# B&R Automation Studio project TD52 (part 144)

#### rtwtypes.h
```c
/********************************************************************
 * COPYRIGHT -- Bernecker + Rainer Industrie-Elektronik Ges.m.b.H.
 ********************************************************************
 * Program: J920_fric
 * File: rtwtypes.h
 * Author: 212348321
 * Created: Mon Jun 13 15:26:38 2016
 ********************************************************************
 * Header for program J920_fric
 ********************************************************************
 * Generated with B&R Automation Studio Target for Simulink V4.2
 * (ERT based)
 ********************************************************************/

#ifndef __RTWTYPES_H__
#define __RTWTYPES_H__
#ifndef TRUE
# define TRUE                          (1U)
#endif

#ifndef FALSE
# define FALSE                         (0U)
#endif

#ifndef __TMWTYPES__
#define __TMWTYPES__
#include <limits.h>

/*=======================================================================*
 * Target hardware information
 *   Device type: Intel->x86/Pentium
 *   Number of bits:     char:   8    short:   16    long:  32
 *                       long:  32
 *                       native word size:  32
 *   Byte ordering: LittleEndian
 *   Signed integer division rounds to: Zero
 *   Shift right on a signed integer as arithmetic shift: on
 *=======================================================================*/

/*=======================================================================*
 * Fixed width word size data types:                                     *
 *   int8_T, int16_T, int32_T     - signed 8, 16, or 32 bit integers     *
 *   uint8_T, uint16_T, uint32_T  - unsigned 8, 16, or 32 bit integers   *
 *   real32_T, real64_T           - 32 and 64 bit floating point numbers *
 *=======================================================================*/
typedef signed char int8_T;
typedef unsigned char uint8_T;
typedef short int16_T;
typedef unsigned short uint16_T;
typedef long int32_T;
typedef unsigned long uint32_T;
typedef float real32_T;
typedef double real64_T;

/*===========================================================================*
 * Generic type definitions: real_T, time_T, boolean_T, int_T, uint_T,       *
 *                           ulong_T, char_T and byte_T.                     *
 *===========================================================================*/
typedef double real_T;
typedef double time_T;
typedef unsigned char boolean_T;
typedef long int_T;
typedef unsigned long uint_T;
typedef unsigned long ulong_T;
typedef char char_T;
typedef unsigned char uchar_T;
typedef char_T byte_T;

/*=======================================================================*
 * Min and Max:                                                          *
 *   int8_T, int16_T, int32_T     - signed 8, 16, or 32 bit integers     *
 *   uint8_T, uint16_T, uint32_T  - unsigned 8, 16, or 32 bit integers   *
 *=======================================================================*/
#define MAX_int8_T                     ((int8_T)(127))
#define MIN_int8_T                     ((int8_T)(-128))
#define MAX_uint8_T                    ((uint8_T)(255U))
#define MIN_uint8_T                    ((uint8_T)(0U))
#define MAX_int16_T                    ((int16_T)(32767))
#define MIN_int16_T                    ((int16_T)(-32768))
#define MAX_uint16_T                   ((uint16_T)(65535U))
#define MIN_uint16_T                   ((uint16_T)(0U))
#define MAX_int32_T                    ((int32_T)(2147483647))
#define MIN_int32_T                    ((int32_T)(-2147483647-1))
#define MAX_uint32_T                   ((uint32_T)(0xFFFFFFFFU))
#define MIN_uint32_T                   ((uint32_T)(0U))

/* Logical type definitions */
#if (!defined(__cplusplus)) && (!defined(__true_false_are_keywords))
#  ifndef false
#   define false                       (0U)
#  endif

#  ifndef true
#   define true                        (1U)
#  endif
#endif

/*
 * Simulink Coder assumes the code is compiled on a target using a 2's complement representation
 * for signed integer values.
 */
#if ((SCHAR_MIN + 1) != -SCHAR_MAX)
#error "This code must be compiled using a 2's complement representation for signed integer values"
#endif

/* This ID is used to detect inclusion of an incompatible rtwtypes.h */
#define RTWTYPES_ID_C08S16I32L32N32F1
#else                                  /* __TMWTYPES__ */
#define TMWTYPES_PREVIOUSLY_INCLUDED
#endif                                 /* __TMWTYPES__ */

/* Block D-Work pointer type */
typedef void * pointer_T;

/* Simulink specific types */
#ifndef __SIMSTRUC_TYPES_H__
#define __SIMSTRUC_TYPES_H__

/* Trigger directions: falling, either, and rising */
typedef enum {
  FALLING_ZERO_CROSSING = -1,
  ANY_ZERO_CROSSING = 0,
  RISING_ZERO_CROSSING = 1
} ZCDirection;

/* Previous state of a trigger signal */
typedef uint8_T ZCSigState;

/* Initial value of a trigger zero crossing signal */
#define UNINITIALIZED_ZCSIG            0x03U
#define NEG_ZCSIG                      0x02U
#define POS_ZCSIG                      0x01U
#define ZERO_ZCSIG                     0x00U

/* Current state of a trigger signal */
typedef enum {
  FALLING_ZCEVENT = -1,
  NO_ZCEVENT = 0,
  RISING_ZCEVENT = 1
} ZCEventType;

#endif                                 /* __SIMSTRUC_TYPES_H__ */
#endif                                 /* __RTWTYPES_H__ */

#ifndef MIN
#define MIN(a,b)                       ((a) < (b) ? (a) : (b))
#endif

#ifndef MAX
#define MAX(a,b)                       ((a) > (b) ? (a) : (b))
#endif
```

#### J920_fric.c
```c
/********************************************************************
 * COPYRIGHT -- Bernecker + Rainer Industrie-Elektronik Ges.m.b.H.
 ********************************************************************
 * Program: J920_fric
 * File: J920_fric.c
 * Author: 212348321
 * Created: Mon Jun 13 15:26:38 2016
 ********************************************************************
 * Implementation of program J920_fric
 ********************************************************************
 * Generated with B&R Automation Studio Target for Simulink V4.2
 * (ERT based)
 ********************************************************************/
#include "J920_fric.h"
#include "J920_fric_private.h"

/*  Defines */

/*  Data Types */

/**************************** GLOBAL DATA *************************************/
/*  Definitions */

/*  Declarations  */

/***************************** FILE SCOPE DATA ********************************/

/*************************** FUNCTIONS ****************************************/

/* Lookup Binary Search Utility BINARYSEARCH_real32_T */
void BINARYSEARCH_real32_T(uint32_T *piLeft, uint32_T *piRght, real32_T u, const
  real32_T *pData, uint32_T iHi, struct fFricIMEP* inst)
{
  /* Find the location of current input value in the data table. */
  *piLeft = 0U;
  *piRght = iHi;
  if (u <= pData[0] ) {
    /* Less than or equal to the smallest point in the table. */
    *piRght = 0U;
  } else if (u >= pData[iHi] ) {
    /* Greater than or equal to the largest point in the table. */
    *piLeft = iHi;
  } else {
    uint32_T i;

    /* Do a binary search. */
    while (( *piRght - *piLeft ) > 1U ) {
      /* Get the average of the left and right indices using to Floor rounding. */
      i = (*piLeft + *piRght) >> 1;

      /* Move either the right index or the left index so that */
      /*  LeftDataPoint <= CurrentValue < RightDataPoint */
      if (u < pData[i] ) {
        *piRght = i;
      } else {
        *piLeft = i;
      }
    }
  }
}

/* Lookup Utility LookUp_real32_T_real32_T */
void LookUp_real32_T_real32_T(real32_T *pY, const real32_T *pYData, real32_T u,
  const real32_T *pUData, uint32_T iHi, struct fFricIMEP* inst)
{
  uint32_T iLeft;
  uint32_T iRght;
  BINARYSEARCH_real32_T( &(iLeft), &(iRght), u, pUData, iHi, inst);

  {
    real32_T lambda;
    if (pUData[iRght] > pUData[iLeft] ) {
      real32_T num;
      real32_T den;
      den = pUData[iRght];
      den = den - pUData[iLeft];
      num = u;
      num = num - pUData[iLeft];
      lambda = num / den;
    } else {
      lambda = 0.0F;
    }

    {
      real32_T yLeftCast;
      real32_T yRghtCast;
      yLeftCast = pYData[iLeft];
      yRghtCast = pYData[iRght];
      yLeftCast += lambda * ( yRghtCast - yLeftCast );
      (*pY) = yLeftCast;
    }
  }
}

/*
 * Output and update for atomic system:
 *    '<S12>/TON'
 *    '<S14>/TON'
 *    '<S16>/TON'
 *    '<S17>/TON'
 */
void J920_fric_TON(boolean_T rtu_IN, real32_T rtu_PT, B_TON_J920_fric *localB,
                   DW_TON_J920_fric *localDW, struct fFricIMEP* inst)
{
  /* local block i/o variables */
  boolean_T rtb_LogicalOperator2_jy;
  boolean_T rtb_RelationalOperator_m;

  /* Logic: '<S20>/Logical Operator2' */
  rtb_LogicalOperator2_jy = !rtu_IN;

  /* DiscreteIntegrator: '<S20>/Discrete-Time Integrator' */
  if (rtb_LogicalOperator2_jy || (localDW->DiscreteTimeIntegrator_PrevRese != 0))
  {
    localDW->DiscreteTimeIntegrator_DSTATE = 0.0F;
  }

  /* RelationalOperator: '<S20>/Relational Operator' incorporates:
   *  DiscreteIntegrator: '<S20>/Discrete-Time Integrator'
   */
  rtb_RelationalOperator_m = (localDW->DiscreteTimeIntegrator_DSTATE >= rtu_PT);

  /* Logic: '<S20>/Logical Operator3' */
  localB->LogicalOperator3 = (rtb_RelationalOperator_m && rtu_IN);

  /* Update for DiscreteIntegrator: '<S20>/Discrete-Time Integrator' incorporates:
   *  DataTypeConversion: '<S29>/Conversion'
   *  Logic: '<S20>/Logical Operator'
   *  Logic: '<S20>/Logical Operator1'
   */
  if (!rtb_LogicalOperator2_jy) {
    localDW->DiscreteTimeIntegrator_DSTATE += (real32_T)
      ((!rtb_RelationalOperator_m) && rtu_IN) * 0.01F;
  }

  if (rtb_LogicalOperator2_jy) {
    localDW->DiscreteTimeIntegrator_PrevRese = 1;
  } else {
    localDW->DiscreteTimeIntegrator_PrevRese = 0;
  }

  /* End of Update for DiscreteIntegrator: '<S20>/Discrete-Time Integrator' */
}

/* Model step function */
void J920_fric_step(B_J920_fric *J920_fric_B, DW_J920_fric *J920_fric_DW,
                    ExtY_J920_fric *J920_fric_Y, struct fFricIMEP* inst)
{
  /* local block i/o variables */
  real32_T rtb_LoadStep_TDly;
  real32_T rtb_ExtDist_TDly;
  real32_T rtb_WGM_TDly;
  real32_T rtb_Vltg_TDly;
  real32_T rtb_rPrChP2s_f;
  real32_T rtb_rPos_Set_WG_Norm_g;
  real32_T rtb_T_EO;
  real32_T rtb_WG_Pos[3];
  real32_T rtb_Comp[3];
  real32_T rtb_P2_IP[10];
  real32_T rtb_PMEP_IP[10];
  real32_T rtb_PMEPCC;
  real32_T rtb_WGCC;
  real32_T rtb_TEO[3];
  real32_T rtb_Comp_j[3];
  real32_T rtb_Comp_d[3];
  real32_T rtb_Sig[3];
  real32_T rtb_Add1_e;
  real32_T rtb_DiscreteTimeIntegrator_n1;
  real32_T rtb_DataTypeConversion_o;
  real32_T rtb_Product_g;
  boolean_T rtb_WGM_reset;
  boolean_T rtb_bVltg_reset;
  boolean_T rtb_LogicalOperator2;
  boolean_T rtb_RelationalOperator;
  boolean_T rtb_LogicalOperator2_e;
  boolean_T rtb_LogicalOperator2_h;
  boolean_T rtb_LogicalOperator_f;
  boolean_T rtb_LogicalOperator1_k;
  boolean_T rtb_Compare;
  boolean_T rtb_Compare_n;
  boolean_T rtb_Compare_h;
  boolean_T rtb_Compare_p;
  real32_T rtb_rTconst_Power_Filt;
  real32_T rtb_WGM_Tconst;
  real32_T rtb_Vltg_Tconst;
  real32_T rtb_DiscreteTimeIntegrator_c;
  boolean_T rtb_RelationalOperator_b;
  real32_T rtb_DiscreteTimeIntegrator_n;
  real32_T rtb_DiscreteTimeIntegrator_p;
  real32_T rtb_DiscreteTimeIntegrator_b;
  real32_T rtb_DiscreteTimeIntegrator_h;
  real32_T rtb_Switch_p;
  boolean_T rtb_LogicalOperator2_m;
  boolean_T rtb_LogicalOperator2_k;
  boolean_T rtb_RelationalOperator2_e;
  real32_T rtb_omega_sensrads;
  real32_T rtb_omega_dot_sensrads2;
  real_T rtb_Divide1;
  boolean_T rtb_LogicalOperator_l[25];
  real_T rtb_multiply[25];
  uint32_T tmp;
  boolean_T rtb_Switch1;
  boolean_T rtb_Switch3;
  real32_T rtb_Add_k;
  real32_T rtb_Product_f;
  real32_T rtb_DiscreteTimeIntegrator;
  real32_T rtb_Sum1;
  real32_T rtb_Product_fm;
  real32_T rtb_Product1_k;
  real32_T rtb_Sum_j;
  int32_T i;
  real_T u;
  real32_T u_0;

  /* S-Function (bur_bus_in): '<Root>/Bus Input1' */
  J920_fric_B->BusInput1 = inst->In;

  /* BusSelector: '<S3>/Bus Selector9' */
  rtb_WGM_reset = J920_fric_B->BusInput1.WGM_reset;
  rtb_bVltg_reset = J920_fric_B->BusInput1.bVltg_reset;

  /* RelationalOperator: '<S28>/Compare' incorporates:
   *  Constant: '<S28>/Constant'
   */
  rtb_Compare = J920_fric_B->BusInput1.bMCBON;

  /* RelationalOperator: '<S27>/Compare' incorporates:
   *  Constant: '<S27>/Constant'
   */
  rtb_Compare_n = !J920_fric_B->BusInput1.bMCBON;

  /* RelationalOperator: '<S24>/Compare' incorporates:
   *  Constant: '<S24>/Constant'
   */
  rtb_Compare_h = J920_fric_B->BusInput1.bGCBON;

  /* RelationalOperator: '<S23>/Compare' incorporates:
   *  Constant: '<S23>/Constant'
   */
  rtb_Compare_p = !J920_fric_B->BusInput1.bGCBON;

  /* Logic: '<S12>/Logical Operator2' incorporates:
   *  Constant: '<S24>/Constant'
   *  Constant: '<S28>/Constant'
   *  Logic: '<S12>/Logical Operator3'
   *  Logic: '<S18>/Logical Operator'
   *  Logic: '<S19>/Logical Operator'
   *  RelationalOperator: '<S21>/FixPt Relational Operator'
   *  RelationalOperator: '<S22>/FixPt Relational Operator'
   *  RelationalOperator: '<S24>/Compare'
   *  RelationalOperator: '<S25>/FixPt Relational Operator'
   *  RelationalOperator: '<S26>/FixPt Relational Operator'
   *  RelationalOperator: '<S28>/Compare'
   *  UnitDelay: '<S21>/Delay Input1'
   *  UnitDelay: '<S22>/Delay Input1'
   *  UnitDelay: '<S25>/Delay Input1'
   *  UnitDelay: '<S26>/Delay Input1'
   */
  rtb_LogicalOperator2 = !(((int32_T)J920_fric_B->BusInput1.bMCBON > (int32_T)
    J920_fric_DW->DelayInput1_DSTATE) || ((int32_T)rtb_Compare_n > (int32_T)
    J920_fric_DW->DelayInput1_DSTATE_k) || (((int32_T)
    J920_fric_B->BusInput1.bGCBON > (int32_T)J920_fric_DW->DelayInput1_DSTATE_h)
    || ((int32_T)rtb_Compare_p > (int32_T)J920_fric_DW->DelayInput1_DSTATE_c)) ||
                           (J920_fric_B->BusInput1.bExt_dist != 0.0F));

  /* S-Function (bur_bus_in): '<Root>/Bus Input' */
  J920_fric_B->BusInput = inst->Para;

  /* BusSelector: '<S3>/Bus Selector4' */
  rtb_LoadStep_TDly = J920_fric_B->BusInput.LoadStep_TDly;
  rtb_rTconst_Power_Filt = J920_fric_B->BusInput.rTconst_Power_Filt;
  rtb_ExtDist_TDly = J920_fric_B->BusInput.ExtDist_TDly;
  rtb_WGM_Tconst = J920_fric_B->BusInput.WGM_Tconst;
  rtb_WGM_TDly = J920_fric_B->BusInput.WGM_TDly;
  rtb_Vltg_Tconst = J920_fric_B->BusInput.Vltg_Tconst;
  rtb_Vltg_TDly = J920_fric_B->BusInput.Vltg_TDly;

  /* Outputs for Atomic SubSystem: '<S12>/TON' */
  J920_fric_TON(rtb_LogicalOperator2, rtb_ExtDist_TDly, &J920_fric_B->TON,
                &J920_fric_DW->TON, inst);

  /* End of Outputs for SubSystem: '<S12>/TON' */

  /* RelationalOperator: '<S14>/Relational Operator' incorporates:
   *  Abs: '<S14>/Abs'
   *  Sum: '<S14>/Add2'
   */
  rtb_RelationalOperator = ((real32_T)fabs(J920_fric_B->BusInput1.Speed -
    J920_fric_B->BusInput.rNEngNom) <= J920_fric_B->BusInput.Speedrange);

  /* Outputs for Atomic SubSystem: '<S14>/TON' */
  J920_fric_TON(rtb_RelationalOperator, rtb_LoadStep_TDly, &J920_fric_B->TON_i,
                &J920_fric_DW->TON_i, inst);

  /* End of Outputs for SubSystem: '<S14>/TON' */

  /* DiscreteIntegrator: '<S32>/Discrete-Time Integrator' */
  if (J920_fric_DW->DiscreteTimeIntegrator_IC_LOADI != 0) {
    J920_fric_DW->DiscreteTimeIntegrator_DSTATE =
      J920_fric_B->BusInput.rIC_Power_filt;
  }

  rtb_DiscreteTimeIntegrator_c = J920_fric_DW->DiscreteTimeIntegrator_DSTATE;

  /* Saturate: '<S15>/Saturation' incorporates:
   *  DiscreteIntegrator: '<S32>/Discrete-Time Integrator'
   */
  if (J920_fric_DW->DiscreteTimeIntegrator_DSTATE >= 0.0F) {
    rtb_DiscreteTimeIntegrator_n = J920_fric_DW->DiscreteTimeIntegrator_DSTATE;
  } else {
    rtb_DiscreteTimeIntegrator_n = 0.0F;
  }

  /* RelationalOperator: '<S15>/Relational Operator' incorporates:
   *  Saturate: '<S15>/Saturation'
   */
  rtb_RelationalOperator_b = (rtb_DiscreteTimeIntegrator_n >=
    J920_fric_B->BusInput.rPower_Thrsh);

  /* DiscreteIntegrator: '<S42>/Discrete-Time Integrator' */
  if (J920_fric_DW->DiscreteTimeIntegrator_IC_LOA_m != 0) {
    J920_fric_DW->DiscreteTimeIntegrator_DSTATE_a = J920_fric_B->BusInput.WGM_y0;
  }

  if (rtb_WGM_reset || (J920_fric_DW->DiscreteTimeIntegrator_PrevRese != 0)) {
    J920_fric_DW->DiscreteTimeIntegrator_DSTATE_a = J920_fric_B->BusInput.WGM_y0;
  }

  rtb_DiscreteTimeIntegrator_n = J920_fric_DW->DiscreteTimeIntegrator_DSTATE_a;

  /* Logic: '<S17>/Logical Operator2' incorporates:
   *  Abs: '<S17>/Abs'
   *  DiscreteIntegrator: '<S42>/Discrete-Time Integrator'
   *  RelationalOperator: '<S17>/Relational Operator1'
   *  Sum: '<S17>/Add'
   */
  rtb_LogicalOperator2_e = !(J920_fric_B->BusInput.WGM_FaultThrsh <= (real32_T)
    fabs(J920_fric_B->BusInput1.rPos_Set_WG_Norm -
         J920_fric_DW->DiscreteTimeIntegrator_DSTATE_a));

  /* Outputs for Atomic SubSystem: '<S17>/TON' */
  J920_fric_TON(rtb_LogicalOperator2_e, rtb_WGM_TDly, &J920_fric_B->TON_n,
                &J920_fric_DW->TON_n, inst);

  /* End of Outputs for SubSystem: '<S17>/TON' */

  /* DiscreteIntegrator: '<S38>/Discrete-Time Integrator' */
  if (J920_fric_DW->DiscreteTimeIntegrator_IC_LOA_l != 0) {
    J920_fric_DW->DiscreteTimeIntegrator_DSTATE_h =
      J920_fric_B->BusInput.Vltg_y0;
  }

  if (rtb_bVltg_reset || (J920_fric_DW->DiscreteTimeIntegrator_PrevRe_f != 0)) {
    J920_fric_DW->DiscreteTimeIntegrator_DSTATE_h =
      J920_fric_B->BusInput.Vltg_y0;
  }

  rtb_DiscreteTimeIntegrator_p = J920_fric_DW->DiscreteTimeIntegrator_DSTATE_h;

  /* DiscreteIntegrator: '<S39>/Discrete-Time Integrator' */
  if (J920_fric_DW->DiscreteTimeIntegrator_IC_LOA_b != 0) {
    J920_fric_DW->DiscreteTimeIntegrator_DSTATE_f =
      J920_fric_B->BusInput.Vltg_y0;
  }

  if (rtb_bVltg_reset || (J920_fric_DW->DiscreteTimeIntegrator_PrevRe_j != 0)) {
    J920_fric_DW->DiscreteTimeIntegrator_DSTATE_f =
      J920_fric_B->BusInput.Vltg_y0;
  }

  rtb_DiscreteTimeIntegrator_b = J920_fric_DW->DiscreteTimeIntegrator_DSTATE_f;

  /* DiscreteIntegrator: '<S40>/Discrete-Time Integrator' */
  if (J920_fric_DW->DiscreteTimeIntegrator_IC_LOA_e != 0) {
    J920_fric_DW->DiscreteTimeIntegrator_DSTATE_o =
      J920_fric_B->BusInput.Vltg_y0;
  }

  if (rtb_bVltg_reset || (J920_fric_DW->DiscreteTimeIntegrator_PrevRe_p != 0)) {
    J920_fric_DW->DiscreteTimeIntegrator_DSTATE_o =
      J920_fric_B->BusInput.Vltg_y0;
  }

  rtb_DiscreteTimeIntegrator_h = J920_fric_DW->DiscreteTimeIntegrator_DSTATE_o;

  /* Sum: '<S36>/Add' incorporates:
   *  DiscreteIntegrator: '<S40>/Discrete-Time Integrator'
   */
  rtb_Product_g = J920_fric_B->BusInput1.U_L3L1 -
    J920_fric_DW->DiscreteTimeIntegrator_DSTATE_o;

  /* Abs: '<S36>/Abs' */
  rtb_Product_g = (real32_T)fabs(rtb_Product_g);

  /* Logic: '<S16>/Logical Operator2' incorporates:
   *  Abs: '<S34>/Abs'
   *  Abs: '<S35>/Abs'
   *  DiscreteIntegrator: '<S38>/Discrete-Time Integrator'
   *  DiscreteIntegrator: '<S39>/Discrete-Time Integrator'
   *  Logic: '<S16>/Logical Operator1'
   *  RelationalOperator: '<S34>/Relational Operator1'
   *  RelationalOperator: '<S35>/Relational Operator1'
   *  RelationalOperator: '<S36>/Relational Operator1'
   *  Sum: '<S34>/Add'
   *  Sum: '<S35>/Add'
   */
  rtb_LogicalOperator2_h = !((J920_fric_B->BusInput.Vltg_FaultThrsh <= (real32_T)
    fabs(J920_fric_B->BusInput1.U_L1L2 -
         J920_fric_DW->DiscreteTimeIntegrator_DSTATE_h)) ||
    (J920_fric_B->BusInput.Vltg_FaultThrsh <= (real32_T)fabs
     (J920_fric_B->BusInput1.U_L2L3 -
      J920_fric_DW->DiscreteTimeIntegrator_DSTATE_f)) ||
    (J920_fric_B->BusInput.Vltg_FaultThrsh <= rtb_Product_g));

  /* Outputs for Atomic SubSystem: '<S16>/TON' */
  J920_fric_TON(rtb_LogicalOperator2_h, rtb_Vltg_TDly, &J920_fric_B->TON_e,
                &J920_fric_DW->TON_e, inst);

  /* End of Outputs for SubSystem: '<S16>/TON' */

  /* Sum: '<S11>/Add1' */
  rtb_Product_g = J920_fric_B->BusInput1.I_L1 - J920_fric_B->BusInput1.I_L2;

  /* Abs: '<S11>/Abs' */
  rtb_Product_g = (real32_T)fabs(rtb_Product_g);

  /* Product: '<S11>/Divide' incorporates:
   *  Constant: '<S11>/Constant'
   *  Sum: '<S11>/Add'
   */
  rtb_Divide1 = (real_T)((J920_fric_B->BusInput1.I_L1 +
    J920_fric_B->BusInput1.I_L2) + J920_fric_B->BusInput1.I_L3) / 9.0;

  /* MinMax: '<S11>/MinMax' */
  if (!(rtb_Divide1 >= 10.0)) {
    rtb_Divide1 = 10.0;
  }

  /* Logic: '<S11>/Logical Operator2' incorporates:
   *  Abs: '<S11>/Abs1'
   *  Logic: '<S11>/Logical Operator'
   *  Logic: '<S11>/Logical Operator1'
   *  MinMax: '<S11>/MinMax'
   *  RelationalOperator: '<S11>/Relational Operator1'
   *  RelationalOperator: '<S11>/Relational Operator2'
   *  Sum: '<S11>/Add2'
   */
  rtb_LogicalOperator2_k = !((((real_T)rtb_Product_g >= rtb_Divide1) || ((real_T)
                               (real32_T)fabs(J920_fric_B->BusInput1.I_L2 -
    J920_fric_B->BusInput1.I_L3) >= rtb_Divide1)) &&
    J920_fric_B->BusInput1.bGCBON);

  /* Sum: '<S13>/Sum of Elements' */
  tmp = (uint32_T)J920_fric_B->BusInput1.bLimpHomeCylG2[0];
  for (i = 0; i < 24; i++) {
    tmp += (uint32_T)J920_fric_B->BusInput1.bLimpHomeCylG2[i + 1];
  }

  /* RelationalOperator: '<S13>/Relational Operator1' incorporates:
   *  Sum: '<S13>/Sum of Elements'
   */
  rtb_LogicalOperator2_m = (18 >= (uint8_T)tmp);

  /* Sum: '<S13>/Sum of Elements1' */
  tmp = (uint32_T)J920_fric_B->BusInput1.bLimpHomeCyl[0];
  for (i = 0; i < 24; i++) {
    tmp += (uint32_T)J920_fric_B->BusInput1.bLimpHomeCyl[i + 1];
  }

  /* RelationalOperator: '<S13>/Relational Operator2' incorporates:
   *  Sum: '<S13>/Sum of Elements1'
   */
  rtb_RelationalOperator2_e = (18 >= (uint8_T)tmp);

  /* Sum: '<S13>/Sum of Elements2' */
  tmp = (uint32_T)J920_fric_B->BusInput1.bLimpHomeCylExt[0];
  for (i = 0; i < 24; i++) {
    tmp += (uint32_T)J920_fric_B->BusInput1.bLimpHomeCylExt[i + 1];
  }

  /* Logic: '<S13>/Logical Operator2' incorporates:
   *  RelationalOperator: '<S13>/Relational Operator3'
   *  Sum: '<S13>/Sum of Elements2'
   */
  rtb_LogicalOperator2_m = (rtb_LogicalOperator2_m && rtb_RelationalOperator2_e &&
                            (18 >= (uint8_T)tmp));

  /* Logic: '<S5>/Logical Operator1' incorporates:
   *  Logic: '<S5>/Logical Operator'
   */
  rtb_RelationalOperator2_e = (J920_fric_B->BusInput1.Man_Cond_On ||
    (J920_fric_B->TON.LogicalOperator3 && J920_fric_B->TON_i.LogicalOperator3 &&
     rtb_RelationalOperator_b && J920_fric_B->TON_n.LogicalOperator3 &&
     J920_fric_B->TON_e.LogicalOperator3 && rtb_LogicalOperator2_k &&
     rtb_LogicalOperator2_m));

  /* Gain: '<S9>/Gain1' */
  rtb_omega_sensrads = 0.104719758F * J920_fric_B->BusInput1.Speed;

  /* DiscreteIntegrator: '<S9>/Filter1' */
  if (J920_fric_DW->Filter1_IC_LOADING != 0) {
    J920_fric_DW->Filter1_DSTATE = J920_fric_B->BusInput.rD0_init;
  }

  if (J920_fric_B->BusInput1.bReset_P_kin) {
    J920_fric_DW->Filter1_DSTATE = J920_fric_B->BusInput.rD0_init;
  }

  /* Product: '<S9>/Filter coefficient N' incorporates:
   *  DiscreteIntegrator: '<S9>/Filter1'
   *  Product: '<S9>/Derivative gain'
   *  Sum: '<S9>/SumD'
   */
  rtb_omega_dot_sensrads2 = (rtb_omega_sensrads * J920_fric_B->BusInput.rD_P_kin
    - J920_fric_DW->Filter1_DSTATE) * J920_fric_B->BusInput.rN_P_kin;

  /* Switch: '<S9>/Switch' incorporates:
   *  Constant: '<S9>/Constant'
   *  Gain: '<S9>/kW//W1'
   *  Logic: '<S9>/Logical Operator'
   *  Logic: '<S9>/Logical Operator1'
   *  Product: '<S9>/Inertia (kgm2)  '
   *  Product: '<S9>/Product1'
   */
  if (!(J920_fric_B->BusInput1.bGCBON && J920_fric_B->BusInput1.bMCBON)) {
    rtb_Switch_p = rtb_omega_dot_sensrads2 * rtb_omega_sensrads *
      J920_fric_B->BusInput.rInertia * 0.001F;
  } else {
    rtb_Switch_p = 0.0F;
  }

  /* End of Switch: '<S9>/Switch' */

  /* Outputs for Atomic SubSystem: '<S47>/Filter' */
  /* DiscreteIntegrator: '<S49>/Discrete-Time Integrator' incorporates:
   *  Delay: '<S7>/Delay'
   */
  if (J920_fric_DW->DiscreteTimeIntegrator_IC_LOA_j != 0) {
    J920_fric_DW->DiscreteTimeIntegrator_DSTATE_e = J920_fric_DW->Delay_DSTATE[0];
  }

  if (J920_fric_DW->DiscreteTimeIntegrator_PrevRe_d != 0) {
    J920_fric_DW->DiscreteTimeIntegrator_DSTATE_e = J920_fric_DW->Delay_DSTATE[0];
  }

  /* Switch: '<S49>/Switch' incorporates:
   *  DiscreteIntegrator: '<S49>/Discrete-Time Integrator'
   */
  rtb_omega_sensrads = J920_fric_DW->DiscreteTimeIntegrator_DSTATE_e;

  /* Update for DiscreteIntegrator: '<S49>/Discrete-Time Integrator' incorporates:
   *  Delay: '<S7>/Delay'
   *  DiscreteIntegrator: '<S49>/Discrete-Time Integrator'
   *  Product: '<S49>/Divide4'
   *  Sum: '<S49>/Sum4'
   */
  J920_fric_DW->DiscreteTimeIntegrator_IC_LOA_j = 0U;
  J920_fric_DW->DiscreteTimeIntegrator_DSTATE_e += (J920_fric_DW->Delay_DSTATE[0]
    - J920_fric_DW->DiscreteTimeIntegrator_DSTATE_e) / 0.2F * 0.01F;
  J920_fric_DW->DiscreteTimeIntegrator_PrevRe_d = 0;

  /* End of Outputs for SubSystem: '<S47>/Filter' */

  /* BusSelector: '<S3>/Bus Selector3' */
  rtb_Product_g = J920_fric_B->BusInput.rP_Nom;

  /* Abs: '<S48>/Abs' */
  rtb_DataTypeConversion_o = (real32_T)fabs(rtb_Product_g);

  /* Switch: '<S48>/Switch' incorporates:
   *  RelationalOperator: '<S48>/Relational Operator'
   */
  if (1.0F >= rtb_DataTypeConversion_o) {
    rtb_Product_g = 1.0F;
  }

  /* End of Switch: '<S48>/Switch' */

  /* Product: '<S47>/Divide' */
  rtb_Product_g = rtb_omega_sensrads / rtb_Product_g;

  /* BusSelector: '<S47>/Bus Selector2' */
  rtb_Comp_d[0] = J920_fric_B->BusInput.PFComp_G_CC.Sig[0];
  rtb_Comp_d[1] = J920_fric_B->BusInput.PFComp_G_CC.Sig[1];
  rtb_Comp_d[2] = J920_fric_B->BusInput.PFComp_G_CC.Sig[2];
  rtb_Sig[0] = J920_fric_B->BusInput.PFComp_G_CC.Comp[0];
  rtb_Sig[1] = J920_fric_B->BusInput.PFComp_G_CC.Comp[1];
  rtb_Sig[2] = J920_fric_B->BusInput.PFComp_G_CC.Comp[2];

  /* Dynamic Look-Up Table Block: '<S47>/PMEP G CC'
   * Input0  Data Type:  Floating Point real32_T
   * Input1  Data Type:  Floating Point real32_T
   * Input2  Data Type:  Floating Point real32_T
   * Output0 Data Type:  Floating Point real32_T
   * Lookup Method: Linear_Endpoint
   *
   */
  LookUp_real32_T_real32_T( &(rtb_DataTypeConversion_o), rtb_Sig, rtb_Product_g,
    rtb_Comp_d, 2U, inst);

  /* BusSelector: '<S3>/Bus Selector8' */
  rtb_Product_g = J920_fric_B->BusInput1.PF_Act;

  /* BusSelector: '<S47>/Bus Selector1' */
  rtb_Sig[0] = J920_fric_B->BusInput.PFComp_CC.Sig[0];
  rtb_Sig[1] = J920_fric_B->BusInput.PFComp_CC.Sig[1];
  rtb_Sig[2] = J920_fric_B->BusInput.PFComp_CC.Sig[2];
  rtb_Comp_d[0] = J920_fric_B->BusInput.PFComp_CC.Comp[0];
  rtb_Comp_d[1] = J920_fric_B->BusInput.PFComp_CC.Comp[1];
  rtb_Comp_d[2] = J920_fric_B->BusInput.PFComp_CC.Comp[2];

  /* Dynamic Look-Up Table Block: '<S47>/PMEP CC'
   * Input0  Data Type:  Floating Point real32_T
   * Input1  Data Type:  Floating Point real32_T
   * Input2  Data Type:  Floating Point real32_T
   * Output0 Data Type:  Floating Point real32_T
   * Lookup Method: Linear_Endpoint
   *
   */
  LookUp_real32_T_real32_T( &(rtb_Add1_e), rtb_Comp_d, rtb_Product_g, rtb_Sig,
    2U, inst);

  /* Sum: '<S47>/Add1' incorporates:
   *  Product: '<S47>/Product'
   *  Product: '<S47>/Product1'
   */
  rtb_Add1_e = rtb_DataTypeConversion_o * rtb_Add1_e * rtb_omega_sensrads +
    rtb_Switch_p;

  /* Switch: '<S53>/Switch1' incorporates:
   *  Constant: '<S53>/Constant1'
   */
  if (J920_fric_B->BusInput1.rPrChP2s != 0.0F) {
    u = J920_fric_B->BusInput1.rPrChP2s;
  } else {
    u = 10.0;
  }

  /* End of Switch: '<S53>/Switch1' */

  /* Switch: '<S53>/Switch' incorporates:
   *  Constant: '<S53>/Constant'
   */
  if (J920_fric_B->BusInput.IMEPVali_Fac != 0.0F) {
    rtb_Divide1 = J920_fric_B->BusInput.IMEPVali_Fac;
  } else {
    rtb_Divide1 = 8.0;
  }

  /* End of Switch: '<S53>/Switch' */

  /* Product: '<S53>/m' */
  rtb_Divide1 *= u;
  for (i = 0; i < 25; i++) {
    /* Logic: '<S8>/Logical Operator' incorporates:
     *  Logic: '<S8>/Logical Operator1'
     *  Logic: '<S8>/Logical Operator2'
     *  RelationalOperator: '<S53>/Relational Operator'
     */
    rtb_Switch1 = !(((real_T)J920_fric_B->BusInput1.rPrIMEP[i] > rtb_Divide1) ||
                    J920_fric_B->BusInput1.bPBCSensErr[i] ||
                    (J920_fric_B->BusInput1.bLimpHomeCylG2[i] ||
                     J920_fric_B->BusInput1.bLimpHomeCyl[i] ||
                     J920_fric_B->BusInput1.bLimpHomeCylExt[i]));

    /* Switch: '<S54>/Switch' incorporates:
     *  Constant: '<S54>/Constant1'
     *  Constant: '<S54>/Constant2'
     *  Constant: '<S56>/Constant'
     *  RelationalOperator: '<S56>/Compare'
     */
    if (J920_fric_B->BusInput1.rPrIMEP[i] < 1.0F) {
      u = -0.2;
    } else {
      u = 0.0;
    }

    /* End of Switch: '<S54>/Switch' */

    /* Product: '<S8>/multiply' incorporates:
     *  Sum: '<S54>/Add'
     */
    rtb_multiply[i] = rtb_Switch1 ? (real_T)J920_fric_B->BusInput1.rPrIMEP[i] +
      u : 0.0;

    /* Logic: '<S8>/Logical Operator' */
    rtb_LogicalOperator_l[i] = rtb_Switch1;
  }

  /* Sum: '<S8>/Sum of Elements' */
  rtb_Divide1 = rtb_multiply[0];

  /* Sum: '<S55>/Sum of Elements1' */
  tmp = (uint32_T)rtb_LogicalOperator_l[0];
  for (i = 0; i < 24; i++) {
    /* Sum: '<S8>/Sum of Elements' */
    rtb_Divide1 += rtb_multiply[i + 1];
    tmp += (uint32_T)rtb_LogicalOperator_l[i + 1];
  }

  /* Sum: '<S55>/Add2' incorporates:
   *  Constant: '<S55>/Constant'
   *  Sum: '<S55>/Add1'
   *  Sum: '<S55>/Add3'
   *  Sum: '<S55>/Sum of Elements1'
   */
  u = (25.0 - (25.0 - (real_T)(uint8_T)tmp)) - (25.0 - (real_T)
    J920_fric_B->BusInput.NumberOfCylinder);

  /* Saturate: '<S55>/Saturation' */
  if (!(u >= 1.0)) {
    u = 1.0;
  }

  /* Product: '<S8>/Divide1' incorporates:
   *  Saturate: '<S55>/Saturation'
   */
  rtb_Divide1 /= u;

  /* DataTypeConversion: '<S8>/Data Type Conversion' */
  rtb_DataTypeConversion_o = (real32_T)rtb_Divide1;

  /* BusSelector: '<S3>/Bus Selector7' */
  rtb_rPrChP2s_f = J920_fric_B->BusInput1.rPrChP2s;
  rtb_rPos_Set_WG_Norm_g = J920_fric_B->BusInput1.rPos_Set_WG_Norm;

  /* Outputs for Atomic SubSystem: '<S3>/PMEP' */
  /* BusSelector: '<S10>/Bus Selector' */
  rtb_WG_Pos[0] = J920_fric_B->BusInput.WGComp_CC.WG_Pos[0];
  rtb_WG_Pos[1] = J920_fric_B->BusInput.WGComp_CC.WG_Pos[1];
  rtb_WG_Pos[2] = J920_fric_B->BusInput.WGComp_CC.WG_Pos[2];
  rtb_Comp[0] = J920_fric_B->BusInput.WGComp_CC.Comp[0];
  rtb_Comp[1] = J920_fric_B->BusInput.WGComp_CC.Comp[1];
  rtb_Comp[2] = J920_fric_B->BusInput.WGComp_CC.Comp[2];

  /* BusSelector: '<S10>/Bus Selector1' */
  for (i = 0; i < 10; i++) {
    rtb_P2_IP[i] = J920_fric_B->BusInput.PMEP_CC.P2_IP[i];
    rtb_PMEP_IP[i] = J920_fric_B->BusInput.PMEP_CC.PMEP_IP[i];
  }

  /* End of BusSelector: '<S10>/Bus Selector1' */
  /* Dynamic Look-Up Table Block: '<S10>/PMEP CC'
   * Input0  Data Type:  Floating Point real32_T
   * Input1  Data Type:  Floating Point real32_T
   * Input2  Data Type:  Floating Point real32_T
   * Output0 Data Type:  Floating Point real32_T
   * Lookup Method: Linear_Endpoint
   *
   */
  LookUp_real32_T_real32_T( &(rtb_PMEPCC), rtb_PMEP_IP, rtb_rPrChP2s_f,
    rtb_P2_IP, 9U, inst);

  /* Dynamic Look-Up Table Block: '<S10>/WG CC'
   * Input0  Data Type:  Floating Point real32_T
   * Input1  Data Type:  Floating Point real32_T
   * Input2  Data Type:  Floating Point real32_T
   * Output0 Data Type:  Floating Point real32_T
   * Lookup Method: Linear_Endpoint
   *
   */
  LookUp_real32_T_real32_T( &(rtb_WGCC), rtb_Comp, rtb_rPos_Set_WG_Norm_g,
    rtb_WG_Pos, 2U, inst);

  /* Product: '<S10>/Product' */
  rtb_Product_f = rtb_PMEPCC * rtb_WGCC;

  /* End of Outputs for SubSystem: '<S3>/PMEP' */

  /* Product: '<S7>/Product' incorporates:
   *  Gain: '<S7>/Gain'
   *  Gain: '<S7>/bar_to_Kpa'
   *  Sum: '<S7>/Subtract1'
   */
  rtb_Product_g = (rtb_DataTypeConversion_o + rtb_Product_f) * 100.0F *
    J920_fric_B->BusInput.NumberOfCylinder * J920_fric_B->BusInput.rEngine_Vd *
    (0.00833333377F * J920_fric_B->BusInput1.Speed);

  /* Sum: '<S7>/Add' */
  rtb_Add_k = rtb_Product_g - rtb_Add1_e;

  /* BusSelector: '<S3>/Bus Selector11' */
  rtb_T_EO = J920_fric_B->BusInput1.T_EO;

  /* BusSelector: '<S3>/Bus Selector5' */
  rtb_omega_sensrads = J920_fric_B->BusInput.rTconst_fricflt_slowfilt;

  /* Outputs for Atomic SubSystem: '<S3>/Fault Detection' */
  /* BusSelector: '<S6>/Bus Selector' */
  rtb_TEO[0] = J920_fric_B->BusInput.TEOComp_CC.TEO[0];
  rtb_TEO[1] = J920_fric_B->BusInput.TEOComp_CC.TEO[1];
  rtb_TEO[2] = J920_fric_B->BusInput.TEOComp_CC.TEO[2];
  rtb_Comp_j[0] = J920_fric_B->BusInput.TEOComp_CC.Comp[0];
  rtb_Comp_j[1] = J920_fric_B->BusInput.TEOComp_CC.Comp[1];
  rtb_Comp_j[2] = J920_fric_B->BusInput.TEOComp_CC.Comp[2];

  /* MATLAB Function: '<S6>/movAvg J920' incorporates:
   *  DataTypeConversion: '<S6>/Data Type Conversion'
   */
  /* MATLAB Function 'IMEP_Based_Fric_Detection/Fault Detection/movAvg J920': '<S46>:1' */
  /*  base 240 --> 20 engine cycle --> 2.4 sec. */
  /* '<S46>:1:10' */
  rtb_Divide1 = J920_fric_DW->y_1 * 359.0 / 360.0 + (real_T)rtb_Add_k / 360.0;

  /* '<S46>:1:11' */
  J920_fric_DW->y_1 = rtb_Divide1;

  /* Logic: '<S6>/Logical Operator' */
  rtb_LogicalOperator_f = !rtb_RelationalOperator2_e;

  /* DiscreteIntegrator: '<S44>/Discrete-Time Integrator' incorporates:
   *  DataTypeConversion: '<S6>/Data Type Conversion1'
   */
  if (J920_fric_DW->DiscreteTimeIntegrator_IC_LO_el != 0) {
    J920_fric_DW->DiscreteTimeIntegrator_DSTATE_g = (real32_T)rtb_Divide1;
  }

  if (rtb_LogicalOperator_f || (J920_fric_DW->DiscreteTimeIntegrator_PrevRe_k !=
       0)) {
    J920_fric_DW->DiscreteTimeIntegrator_DSTATE_g = (real32_T)rtb_Divide1;
  }

  rtb_DiscreteTimeIntegrator = J920_fric_DW->DiscreteTimeIntegrator_DSTATE_g;

  /* Sum: '<S44>/Sum1' incorporates:
   *  DiscreteIntegrator: '<S44>/Discrete-Time Integrator'
   */
  rtb_Sum1 = rtb_Add_k - J920_fric_DW->DiscreteTimeIntegrator_DSTATE_g;

  /* End of Outputs for SubSystem: '<S3>/Fault Detection' */

  /* BusSelector: '<S3>/Bus Selector5' */
  u_0 = J920_fric_B->BusInput.rTconst_fricflt_fastfilt;

  /* Outputs for Atomic SubSystem: '<S3>/Fault Detection' */
  /* Logic: '<S6>/Logical Operator1' */
  rtb_LogicalOperator1_k = !rtb_RelationalOperator2_e;

  /* Dynamic Look-Up Table Block: '<S6>/TEO CC'
   * Input0  Data Type:  Floating Point real32_T
   * Input1  Data Type:  Floating Point real32_T
   * Input2  Data Type:  Floating Point real32_T
   * Output0 Data Type:  Floating Point real32_T
   * Lookup Method: Linear_Endpoint
   *
   */
  LookUp_real32_T_real32_T( &(rtb_DiscreteTimeIntegrator_n1), rtb_Comp_j,
    rtb_T_EO, rtb_TEO, 2U, inst);

  /* Product: '<S6>/Product' */
  rtb_Product_fm = rtb_DiscreteTimeIntegrator_n1 *
    J920_fric_B->BusInput.Diff_Thrsh;

  /* Product: '<S6>/Product1' */
  rtb_Product1_k = rtb_DiscreteTimeIntegrator_n1 *
    J920_fric_B->BusInput.Abs_Thrsh;

  /* DiscreteIntegrator: '<S45>/Discrete-Time Integrator' incorporates:
   *  DataTypeConversion: '<S6>/Data Type Conversion1'
   */
  if (J920_fric_DW->DiscreteTimeIntegrator_IC_LO_jk != 0) {
    J920_fric_DW->DiscreteTimeIntegrator_DSTATE_p = (real32_T)rtb_Divide1;
  }

  if (rtb_LogicalOperator1_k || (J920_fric_DW->DiscreteTimeIntegrator_PrevR_dw
       != 0)) {
    J920_fric_DW->DiscreteTimeIntegrator_DSTATE_p = (real32_T)rtb_Divide1;
  }

  rtb_DiscreteTimeIntegrator_n1 = J920_fric_DW->DiscreteTimeIntegrator_DSTATE_p;

  /* End of DiscreteIntegrator: '<S45>/Discrete-Time Integrator' */

  /* Sum: '<S6>/Sum' */
  rtb_Sum_j = rtb_DiscreteTimeIntegrator - rtb_DiscreteTimeIntegrator_n1;

  /* Switch: '<S6>/Switch1' incorporates:
   *  Constant: '<S6>/3'
   *  Constant: '<S6>/6'
   *  RelationalOperator: '<S6>/Relational Operator1'
   *  RelationalOperator: '<S6>/Relational Operator2'
   *  Switch: '<S6>/Switch3'
   */
  if (rtb_RelationalOperator2_e) {
    rtb_Switch1 = (rtb_Product1_k <= rtb_DiscreteTimeIntegrator);
    rtb_Switch3 = (rtb_Product_fm <= rtb_Sum_j);
  } else {
    rtb_Switch1 = FALSE;
    rtb_Switch3 = FALSE;
  }

  /* End of Switch: '<S6>/Switch1' */

  /* Update for DiscreteIntegrator: '<S44>/Discrete-Time Integrator' incorporates:
   *  Product: '<S44>/Divide'
   */
  J920_fric_DW->DiscreteTimeIntegrator_IC_LO_el = 0U;
  if (!rtb_LogicalOperator_f) {
    /* Saturate: '<S44>/Saturation' */
    if (!(u_0 >= 1.0F)) {
      u_0 = 1.0F;
    }

    /* End of Saturate: '<S44>/Saturation' */
    J920_fric_DW->DiscreteTimeIntegrator_DSTATE_g += rtb_Sum1 / u_0 * 0.01F;
  }

  if (rtb_LogicalOperator_f) {
    J920_fric_DW->DiscreteTimeIntegrator_PrevRe_k = 1;
  } else {
    J920_fric_DW->DiscreteTimeIntegrator_PrevRe_k = 0;
  }

  /* End of Update for DiscreteIntegrator: '<S44>/Discrete-Time Integrator' */

  /* Update for DiscreteIntegrator: '<S45>/Discrete-Time Integrator' incorporates:
   *  Product: '<S45>/Divide'
   *  Saturate: '<S45>/Saturation'
   *  Sum: '<S45>/Sum1'
   */
  J920_fric_DW->DiscreteTimeIntegrator_IC_LO_jk = 0U;
  if (!rtb_LogicalOperator1_k) {
    /* Saturate: '<S45>/Saturation' */
    if (!(rtb_omega_sensrads >= 1.0F)) {
      rtb_omega_sensrads = 1.0F;
    }

    J920_fric_DW->DiscreteTimeIntegrator_DSTATE_p += (rtb_Add_k -
      rtb_DiscreteTimeIntegrator_n1) / rtb_omega_sensrads * 0.01F;
  }

  if (rtb_LogicalOperator1_k) {
    J920_fric_DW->DiscreteTimeIntegrator_PrevR_dw = 1;
  } else {
    J920_fric_DW->DiscreteTimeIntegrator_PrevR_dw = 0;
  }

  /* End of Update for DiscreteIntegrator: '<S45>/Discrete-Time Integrator' */
  /* End of Outputs for SubSystem: '<S3>/Fault Detection' */

  /* BusCreator: '<S3>/Bus Creator1' */
  J920_fric_Y->OUT.Fault_Abs = rtb_Switch1;
  J920_fric_Y->OUT.Fault_Diff = rtb_Switch3;

  /* Product: '<S7>/Product1' */
  rtb_omega_sensrads = J920_fric_B->BusInput.NumberOfCylinder *
    J920_fric_B->BusInput.rEngine_Vd * J920_fric_B->BusInput1.Speed;

  /* Saturate: '<S7>/Saturation' */
  if (!(rtb_omega_sensrads >= 1.0F)) {
    rtb_omega_sensrads = 1.0F;
  }

  /* End of Saturate: '<S7>/Saturation' */

  /* BusCreator: '<S3>/Bus Creator' incorporates:
   *  Gain: '<S7>/Gain1'
   *  Gain: '<S7>/Gain2'
   *  Gain: '<S7>/Gain3'
   *  Gain: '<S7>/Gain4'
   *  Product: '<S7>/Divide'
   *  Product: '<S7>/Divide1'
   *  SignalConversion: '<S3>/TmpSignal ConversionAtBus CreatorInport16'
   *  SignalConversion: '<S3>/TmpSignal ConversionAtBus CreatorInport5'
   *  SignalConversion: '<S3>/TmpSignal ConversionAtBus CreatorInport6'
   */
  J920_fric_Y->dbg.Pfric = rtb_Add_k;
  J920_fric_Y->dbg.P_kin = rtb_Switch_p;
  J920_fric_Y->dbg.omega_dot = rtb_omega_dot_sensrads2;
  J920_fric_Y->dbg.Power = rtb_DiscreteTimeIntegrator_c;
  J920_fric_Y->dbg.FD_Param_Diff[0] = rtb_Sum_j;
  J920_fric_Y->dbg.FD_Param_Diff[1] = rtb_Product_fm;
  J920_fric_Y->dbg.FD_Param_Abs[0] = rtb_DiscreteTimeIntegrator;
  J920_fric_Y->dbg.FD_Param_Abs[1] = rtb_Product1_k;
  J920_fric_Y->dbg.BMEP = 1.0F / rtb_omega_sensrads * (120.0F * rtb_Add1_e) *
    0.01F;
  J920_fric_Y->dbg.PMEP = rtb_Product_f;
  J920_fric_Y->dbg.IMEP_avg = rtb_DataTypeConversion_o;
  J920_fric_Y->dbg.Pmech = rtb_Add1_e;
  J920_fric_Y->dbg.Condition_ON = rtb_RelationalOperator2_e;
  J920_fric_Y->dbg.Pind = rtb_Product_g;
  J920_fric_Y->dbg.FMEP = 120.0F * rtb_Add_k / rtb_omega_sensrads * 0.01F;
  J920_fric_Y->dbg.Pact = J920_fric_B->BusInput1.Pact;
  J920_fric_Y->dbg.Speed = J920_fric_B->BusInput1.Speed;
  J920_fric_Y->dbg.Condition_dbg[0] = J920_fric_B->TON.LogicalOperator3;
  J920_fric_Y->dbg.Condition_dbg[1] = J920_fric_B->TON_i.LogicalOperator3;
  J920_fric_Y->dbg.Condition_dbg[2] = rtb_RelationalOperator_b;
  J920_fric_Y->dbg.Condition_dbg[3] = J920_fric_B->TON_n.LogicalOperator3;
  J920_fric_Y->dbg.Condition_dbg[4] = J920_fric_B->TON_e.LogicalOperator3;
  J920_fric_Y->dbg.Condition_dbg[5] = rtb_LogicalOperator2_k;
  J920_fric_Y->dbg.Condition_dbg[6] = rtb_LogicalOperator2_m;

  /* S-Function (bur_bus_out): '<Root>/Bus Output' */
  inst->Out = J920_fric_Y->OUT;

  /* S-Function (bur_bus_out): '<Root>/Bus Output1' */
  inst->dbgOut = J920_fric_Y->dbg;

  /* Sum: '<S32>/Sum' */
  rtb_Switch_p = J920_fric_B->BusInput1.Pact - rtb_DiscreteTimeIntegrator_c;

  /* Sum: '<S38>/Sum' */
  rtb_Product_fm = J920_fric_B->BusInput1.U_L1L2 - rtb_DiscreteTimeIntegrator_p;

  /* Sum: '<S39>/Sum' */
  rtb_Add_k = J920_fric_B->BusInput1.U_L2L3 - rtb_DiscreteTimeIntegrator_b;

  /* Sum: '<S40>/Sum' */
  rtb_Product_f = J920_fric_B->BusInput1.U_L3L1 - rtb_DiscreteTimeIntegrator_h;

  /* Sum: '<S42>/Sum' */
  rtb_Sum1 = J920_fric_B->BusInput1.rPos_Set_WG_Norm -
    rtb_DiscreteTimeIntegrator_n;

  /* UnitDelay: '<S4>/Unit Delay' */
  J920_fric_B->UnitDelay = J920_fric_DW->UnitDelay_DSTATE;

  /* S-Function (bur_out): '<Root>/Output8' */
  inst->Info = J920_fric_B->UnitDelay;

  /* Update for UnitDelay: '<S26>/Delay Input1' */
  J920_fric_DW->DelayInput1_DSTATE = rtb_Compare;

  /* Update for UnitDelay: '<S25>/Delay Input1' */
  J920_fric_DW->DelayInput1_DSTATE_k = rtb_Compare_n;

  /* Update for UnitDelay: '<S22>/Delay Input1' */
  J920_fric_DW->DelayInput1_DSTATE_h = rtb_Compare_h;

  /* Update for UnitDelay: '<S21>/Delay Input1' */
  J920_fric_DW->DelayInput1_DSTATE_c = rtb_Compare_p;

  /* Update for DiscreteIntegrator: '<S32>/Discrete-Time Integrator' */
  J920_fric_DW->DiscreteTimeIntegrator_IC_LOADI = 0U;

  /* Saturate: '<S32>/Saturation' */
  if (!(rtb_rTconst_Power_Filt >= 1.0F)) {
    rtb_rTconst_Power_Filt = 1.0F;
  }

  /* End of Saturate: '<S32>/Saturation' */

  /* Update for DiscreteIntegrator: '<S32>/Discrete-Time Integrator' incorporates:
   *  Product: '<S32>/Divide'
   */
  J920_fric_DW->DiscreteTimeIntegrator_DSTATE += rtb_Switch_p /
    rtb_rTconst_Power_Filt * 0.01F;

  /* Update for DiscreteIntegrator: '<S42>/Discrete-Time Integrator' incorporates:
   *  Product: '<S42>/Divide'
   */
  J920_fric_DW->DiscreteTimeIntegrator_IC_LOA_m = 0U;
  if (!rtb_WGM_reset) {
    /* Saturate: '<S42>/Saturation' */
    if (!(rtb_WGM_Tconst >= 0.01F)) {
      rtb_WGM_Tconst = 0.01F;
    }

    /* End of Saturate: '<S42>/Saturation' */
    J920_fric_DW->DiscreteTimeIntegrator_DSTATE_a += rtb_Sum1 / rtb_WGM_Tconst *
      0.01F;
  }

  if (rtb_WGM_reset) {
    J920_fric_DW->DiscreteTimeIntegrator_PrevRese = 1;
  } else {
    J920_fric_DW->DiscreteTimeIntegrator_PrevRese = 0;
  }

  /* End of Update for DiscreteIntegrator: '<S42>/Discrete-Time Integrator' */

  /* Update for DiscreteIntegrator: '<S38>/Discrete-Time Integrator' incorporates:
   *  Product: '<S38>/Divide'
   */
  J920_fric_DW->DiscreteTimeIntegrator_IC_LOA_l = 0U;
  if (!rtb_bVltg_reset) {
    /* Saturate: '<S38>/Saturation' */
    if (rtb_Vltg_Tconst >= 0.01F) {
      rtb_DiscreteTimeIntegrator_n = rtb_Vltg_Tconst;
    } else {
      rtb_DiscreteTimeIntegrator_n = 0.01F;
    }

    /* End of Saturate: '<S38>/Saturation' */
    J920_fric_DW->DiscreteTimeIntegrator_DSTATE_h += rtb_Product_fm /
      rtb_DiscreteTimeIntegrator_n * 0.01F;
  }

  if (rtb_bVltg_reset) {
    J920_fric_DW->DiscreteTimeIntegrator_PrevRe_f = 1;
  } else {
    J920_fric_DW->DiscreteTimeIntegrator_PrevRe_f = 0;
  }

  /* End of Update for DiscreteIntegrator: '<S38>/Discrete-Time Integrator' */

  /* Update for DiscreteIntegrator: '<S39>/Discrete-Time Integrator' incorporates:
   *  Product: '<S39>/Divide'
   */
  J920_fric_DW->DiscreteTimeIntegrator_IC_LOA_b = 0U;
  if (!rtb_bVltg_reset) {
    /* Saturate: '<S39>/Saturation' */
    if (rtb_Vltg_Tconst >= 0.01F) {
      rtb_DiscreteTimeIntegrator_n = rtb_Vltg_Tconst;
    } else {
      rtb_DiscreteTimeIntegrator_n = 0.01F;
    }

    /* End of Saturate: '<S39>/Saturation' */
    J920_fric_DW->DiscreteTimeIntegrator_DSTATE_f += rtb_Add_k /
      rtb_DiscreteTimeIntegrator_n * 0.01F;
  }

  if (rtb_bVltg_reset) {
    J920_fric_DW->DiscreteTimeIntegrator_PrevRe_j = 1;
  } else {
    J920_fric_DW->DiscreteTimeIntegrator_PrevRe_j = 0;
  }

  /* End of Update for DiscreteIntegrator: '<S39>/Discrete-Time Integrator' */

  /* Update for DiscreteIntegrator: '<S40>/Discrete-Time Integrator' incorporates:
   *  Product: '<S40>/Divide'
   */
  J920_fric_DW->DiscreteTimeIntegrator_IC_LOA_e = 0U;
  if (!rtb_bVltg_reset) {
    /* Saturate: '<S40>/Saturation' */
    if (!(rtb_Vltg_Tconst >= 0.01F)) {
      rtb_Vltg_Tconst = 0.01F;
    }

    /* End of Saturate: '<S40>/Saturation' */
    J920_fric_DW->DiscreteTimeIntegrator_DSTATE_o += rtb_Product_f /
      rtb_Vltg_Tconst * 0.01F;
  }

  if (rtb_bVltg_reset) {
    J920_fric_DW->DiscreteTimeIntegrator_PrevRe_p = 1;
  } else {
    J920_fric_DW->DiscreteTimeIntegrator_PrevRe_p = 0;
  }

  /* End of Update for DiscreteIntegrator: '<S40>/Discrete-Time Integrator' */

  /* Update for DiscreteIntegrator: '<S9>/Filter1' */
  J920_fric_DW->Filter1_IC_LOADING = 0U;
  J920_fric_DW->Filter1_DSTATE += 0.01F * rtb_omega_dot_sensrads2;

  /* Update for Delay: '<S7>/Delay' */
  J920_fric_DW->Delay_DSTATE[0] = J920_fric_DW->Delay_DSTATE[1];
  J920_fric_DW->Delay_DSTATE[1] = J920_fric_B->BusInput1.Pact;

  /* Update for UnitDelay: '<S4>/Unit Delay' */
  J920_fric_DW->UnitDelay_DSTATE = 71U;
}

/* Model initialize function */
void J920_fric_initialize(DW_J920_fric *J920_fric_DW, struct fFricIMEP* inst)
{
  /* InitializeConditions for DiscreteIntegrator: '<S32>/Discrete-Time Integrator' */
  J920_fric_DW->DiscreteTimeIntegrator_IC_LOADI = 1U;

  /* InitializeConditions for DiscreteIntegrator: '<S42>/Discrete-Time Integrator' */
  J920_fric_DW->DiscreteTimeIntegrator_IC_LOA_m = 1U;

  /* InitializeConditions for DiscreteIntegrator: '<S38>/Discrete-Time Integrator' */
  J920_fric_DW->DiscreteTimeIntegrator_IC_LOA_l = 1U;

  /* InitializeConditions for DiscreteIntegrator: '<S39>/Discrete-Time Integrator' */
  J920_fric_DW->DiscreteTimeIntegrator_IC_LOA_b = 1U;

  /* InitializeConditions for DiscreteIntegrator: '<S40>/Discrete-Time Integrator' */
  J920_fric_DW->DiscreteTimeIntegrator_IC_LOA_e = 1U;

  /* InitializeConditions for DiscreteIntegrator: '<S9>/Filter1' */
  J920_fric_DW->Filter1_IC_LOADING = 1U;

  /* InitializeConditions for Atomic SubSystem: '<S47>/Filter' */
  /* InitializeConditions for DiscreteIntegrator: '<S49>/Discrete-Time Integrator' */
  J920_fric_DW->DiscreteTimeIntegrator_IC_LOA_j = 1U;

  /* End of InitializeConditions for SubSystem: '<S47>/Filter' */

  /* InitializeConditions for Atomic SubSystem: '<S3>/Fault Detection' */
  /* InitializeConditions for DiscreteIntegrator: '<S44>/Discrete-Time Integrator' */
  J920_fric_DW->DiscreteTimeIntegrator_IC_LO_el = 1U;

  /* InitializeConditions for DiscreteIntegrator: '<S45>/Discrete-Time Integrator' */
  J920_fric_DW->DiscreteTimeIntegrator_IC_LO_jk = 1U;

  /* End of InitializeConditions for SubSystem: '<S3>/Fault Detection' */
}

/* Model terminate function */
void J920_fric_terminate(struct fFricIMEP* inst)
{
  /* (no terminate code required) */
}

/*======================== TOOL VERSION INFORMATION ==========================*
 * MATLAB 8.0 (R2012b)20-Jul-2012                                             *
 * Simulink 8.0 (R2012b)20-Jul-2012                                           *
 * Simulink Coder 8.3 (R2012b)20-Jul-2012                                     *
 * Embedded Coder 6.3 (R2012b)20-Jul-2012                                     *
 * Stateflow 8.0 (R2012b)20-Jul-2012                                          *
 *============================================================================*/

/*======================= LICENSE IN USE INFORMATION =========================*
 * matlab                                                                     *
 * matlab_coder                                                               *
 * real-time_workshop                                                         *
 * rtw_embedded_coder                                                         *
 * simulink                                                                   *
 *============================================================================*/
```

#### fFricIMEP.c
```c
/********************************************************************
 * COPYRIGHT -- Bernecker + Rainer Industrie-Elektronik Ges.m.b.H.
 ********************************************************************
 * Program: J920_fric
 * File: fFricIMEP.c
 * Author: 212348321
 * Created: Mon Jun 13 15:26:38 2016
 ********************************************************************
 * Implementation of program J920_fric
 ********************************************************************
 * Generated with B&R Automation Studio Target for Simulink V4.2
 * (ERT based)
 ********************************************************************/
#include <bur/plctypes.h>
#include "J920_fric.h"
#include "rtwtypes.h"

/* Defines */
#define SS_TERMINATE 4
#define SS_OUTPUT 3
#define SS_INITIALIZE 2

/*  Data Types */

/**************************** GLOBAL DATA *************************************/
/*  Definitions */

/*  Declarations  */

/***************************** FILE SCOPE DATA ********************************/

/*************************** FUNCTIONS ****************************************/
#ifdef __cplusplus

unsigned long bur_heap_size = 6553500;

#endif

void fFricIMEP(struct fFricIMEP* inst)
{
  B_J920_fric *J920_fric_B = &(inst)->bur_B_J920_fric;
	DW_J920_fric *J920_fric_DW = &(inst)->bur_DW_J920_fric;
	ExtY_J920_fric *J920_fric_Y = &(inst)->bur_ExtY_J920_fric;

  switch (inst->ssMethodType)
  {
   case SS_INITIALIZE:
    /* call model initialize function */
    J920_fric_initialize(J920_fric_DW, inst);
    break;

   case SS_OUTPUT:
    /* call model step function */
    J920_fric_step(J920_fric_B, J920_fric_DW, J920_fric_Y, inst);

    break;

   case SS_TERMINATE:
    /* call model terminate function */
    J920_fric_terminate(inst);
    break;
  }
}

/*****************************************************************************
   Function block sample time: 0.01s
 *****************************************************************************/

/*****************************************************************************
   B&R Automation Studio Target for Simulink Version: A4.5.1 (27-Jul-2015)
 *****************************************************************************/

/*======================== TOOL VERSION INFORMATION ==========================*
 * MATLAB 8.0 (R2012b)20-Jul-2012                                             *
 * Simulink 8.0 (R2012b)20-Jul-2012                                           *
 * Simulink Coder 8.3 (R2012b)20-Jul-2012                                     *
 * Embedded Coder 6.3 (R2012b)20-Jul-2012                                     *
 * Stateflow 8.0 (R2012b)20-Jul-2012                                          *
 *============================================================================*/

/*======================= LICENSE IN USE INFORMATION =========================*
 * matlab                                                                     *
 * matlab_coder                                                               *
 * real-time_workshop                                                         *
 * rtw_embedded_coder                                                         *
 * simulink                                                                   *
 *============================================================================*/
```

#### lib_properties.txt
```
For manual assignment to hardware configuration please
add the following additional include directories:

\Logical\MATLAB_includes\R2012b\

And the following additional build options:

-lm -D MODEL=J920_fric -D NUMST=1 -D NCSTATES=0 -D HAVESTDIO -D ONESTEPFCN=1 -D TERMFCN=1 -D MAT_FILE=0 -D MULTI_INSTANCE_CODE=1 -D INTEGER_CODE=0 -D MT=0 -D CLASSIC_INTERFACE=0 -D TID01EQ=0
```

### Program Logical/CBM/IN_CBM (IEC, version 4.12.0) - Program

#### IN_CBM.st - Implementation code
```iecst
(*******************************************************************************
AGGR: IN CBM

This code is confidential AND proprietary to the INNIO Company.
It may NOT be used in any form, or reproduced in any manner, without the express
written permission of the INNIO Company.
Copyright, INNIO Company, 2022

Customized modifications: -
------------------------
History:
-------
V4.06.01 	30-07-2018 	502423184		header added, added rCA_MFBxx
			13-11-2018	502423184		added new times stamp to replace clock_ms()
V4.12.00	08-09-2022	Andre			Select the engine speed from the ICxx module also if SEMIC is active

Instructions FOR use:
--------------------
- use in a 10ms cycle time

Outstandings:
------------
-

*******************************************************************************)
PROGRAM _INIT
(** A: GE Prop info *)
	strGEProp			:=	'';
	strcat(ADR(strGEProp),ADR('The information contained in this document and any documents attached hereto is privileged or confidential.$n'));
	strcat(ADR(strGEProp),ADR('It is the property of INNIO Company and shall not be used, disclosed to others,$n'));
	strcat(ADR(strGEProp),ADR('or reproduced without the express written consent of INNIO Company.$n'));
	strLine				:=	'$n';
(** B: HMI Speed *)
	tiHMI_Delay			:=	T#10m; 		//Depends on HMI Version

END_PROGRAM

PROGRAM _CYCLIC

(** 0: test development *)
	IF bTEST THEN
		IN_CB.iSt_OpMode	:=	50 * 65536;	//NetP
		rN_Eng				:=	1000;		//Speed
		bGnlTrip			:=	FALSE;
		bGnlTrip1			:=	FALSE;
		bGnlTrip2			:=	FALSE;
		bGnlTrip3			:=	FALSE;
		TON_PBC_Man_Trig.IN	:=	NOT VIS2MM.ECB.bTrig AND NOT bPBC_Write AND NOT xOpMode.Stop;
		TON_PBC_Man_Trig.PT	:=	T#15m;
		TON_PBC_Man_Trig();
		IF EDGEPOS(TON_PBC_Man_Trig.Q) THEN
			VIS2MM.ECB.bTrig	:= bTest2;
		END_IF
	END_IF

(** 1: get engine type *)
	xEngType.Motortype := Para.iEng_Motortype;
	xEngType();

(** 2: get operation mode *)
	xOpMode.in			:=	IN_CB.iSt_OpMode;
	xOpMode();

(** 3: Engine speed measured 1/min *)
	IF Para.b_IgnIC_900Active OR Para.bSEMIC_Active THEN
		rN_Eng := IN_CB.rN_IgnIC_Act;
	ELSIF Para.bSA_Ign_Active THEN
		rN_Eng := IN_CB.rN_IgnSAFI_Act;
	END_IF;

(** 4: set engine cycle bit *) //bit is TRUE when engine is in a new cycle
	rCnt_N				:=	rCnt_N + rN_Eng / 60 / 100; (* convert rpm to rounds per 10ms *)
	IF rCnt_N >= 2.0 THEN	(* 4 stroke engine *)
		bNewEngCycle	:=	TRUE;
		rCnt_N			:=	rCnt_N - 2.0;
		bPBC_NewData	:=	TRUE;	(* trigger new data for pbc buffering *)
	ELSE
		bNewEngCycle	:=	FALSE;
	END_IF

(** 5: get time *)
	DTGetTime_RPS(enable:=1);
	DT_TO_DTStructure(DTGetTime_RPS.DT1, ADR(tRealTime));
	tTimeStamp.Year		:=	UINT_TO_USINT(tRealTime.year MOD 100);
	tTimeStamp.Month	:=	tRealTime.month;
	tTimeStamp.Day		:=	tRealTime.day;
	tTimeStamp.Hour		:=	tRealTime.hour;
	tTimeStamp.Minute	:=	tRealTime.minute;
	IF tTimeStamp.Second <> tRealTime.second THEN
		iMilliSec	:=	0;
	ELSE
		iMilliSec	:=	MIN(iMilliSec + 10,990);
	END_IF
	tTimeStamp.Second	:=	tRealTime.second;

	iSec	:=	USINT_TO_UDINT(tRealTime.second);
	iMin	:=	USINT_TO_UDINT(tRealTime.minute);
	iHour	:=	USINT_TO_UDINT(tRealTime.hour);

	iSec	:=	iSec MOD 60;
	iMin	:=	iMin MOD 60;
	iHour	:=	iHour MOD 24;

	tiStamp	:=	UDINT_TO_TIME(
					iHour	* 60 * 60 * 1000 +
					iMin	* 60 * 1000 +
					iSec	* 1000 +
					iMilliSec
				);
	IF tiStamp = T#0ms THEN
		tiStamp	:=	T#24h;
	END_IF

(** 6: convert data from SAFI *)
	FOR iIdx_Cyl:= 1 TO xEngType.NumberOfCylinder/2 DO
		IF Para.bSA_PBC_Active THEN
			(* speed measuring with DMR function*)
			IF IN_CB.tMS_PBC0[iIdx_Cyl].data1 <> 16#7FFF THEN rN_SAFI[iIdx_Cyl * 2 - 1]		:= UINT_TO_REAL(IN_CB.tMS_PBC0[iIdx_Cyl].data1)/10; END_IF
			IF IN_CB.tMS_PBC1[iIdx_Cyl].data1 <> 16#7FFF THEN rN_SAFI[iIdx_Cyl * 2]			:= UINT_TO_REAL(IN_CB.tMS_PBC1[iIdx_Cyl].data1)/10; END_IF
			(* PBC14 and PBC15 *)		(* data2 *)
			rCA_MFB10[iIdx_Cyl * 2 - 1]		:= INT_TO_REAL(UINT_TO_INT(IN_CB.tMS_PBC14[iIdx_Cyl].data2))/10;		(*convert from 0.1CA to 1CA*)
			rCA_MFB10[iIdx_Cyl * 2]			:= INT_TO_REAL(UINT_TO_INT(IN_CB.tMS_PBC15[iIdx_Cyl].data2))/10;
			(* PBC14 and PBC15 *)		(* data3 *)
			rCA_MFB90[iIdx_Cyl * 2 - 1]		:= INT_TO_REAL(UINT_TO_INT(IN_CB.tMS_PBC14[iIdx_Cyl].data3))/10;		(*convert from 0.1CA to 1CA*)
			rCA_MFB90[iIdx_Cyl * 2]			:= INT_TO_REAL(UINT_TO_INT(IN_CB.tMS_PBC15[iIdx_Cyl].data3))/10;
		ELSE
			(* speed measuring with KLS function*)
			IF IN_CB.KLS_md00[iIdx_Cyl].data1 <> 16#7FFF THEN rN_SAFI[iIdx_Cyl * 2 - 1]	 	:= UINT_TO_REAL(IN_CB.KLS_md00[iIdx_Cyl].data1)/10; END_IF
			IF IN_CB.KLS_md01[iIdx_Cyl].data1 <> 16#7FFF THEN rN_SAFI[iIdx_Cyl * 2]			:= UINT_TO_REAL(IN_CB.KLS_md01[iIdx_Cyl].data1)/10; END_IF
		END_IF
	END_FOR

END_PROGRAM
```

#### IN_CBM.var - Local variables
```iecst
(********************************************************************
 * COPYRIGHT -- INNIO Company
 ********************************************************************
 * Program: CBM_TEST
 * File: CBM_TEST.var
 * Author: 502293141
 * Created: February 20, 2015
 ********************************************************************
 * Local variables of program CBM_TEST
 ********************************************************************)
VAR
	DTGetTime_RPS : DTGetTime;
	TON_PBC_Man_Trig : TON;
	rCnt_N : REAL;
	bTest2 : BOOL := 0;
	iIdx_Cyl : USINT;
	iMilliSec : UDINT;
	iSec : UDINT;
	iHour : UDINT;
	iMin : UDINT;
END_VAR
```

### Program Logical/CBM/MsgCB (IEC) - + Messages

- MsgCBCyclic.st (not readable text: treated as protected, skipped)

- MsgCBInit.st (not readable text: treated as protected, skipped)

#### MsgCB.var
```iecst
VAR
	iAdrAmmBase2MM : UDINT;
	iAdrMM2AmmBase : UDINT;
	xMsg2308 : Msg;
	xMsg2293 : Msg;
	xMsg9223 : Msg;
	xTP_FMEP_Fault_Dtct_Save : TP_10ms := (0);
	xMsg2926 : Msg;	(** B2926: ATD has further information *)
END_VAR
```

### Program Logical/CBM/ParCB (IEC, version 4.06.0) - + Parameter handling

- perm_par.st (not readable text: treated as protected, skipped)

#### perm_par.var
```iecst
VAR
	tParaIntern : ParaHandler_typ; (*Connector type to perm_par*)
	tMM2ParaBase_ReadBack : MM2ParaBase_type; (*INTERNAL! V4.06 new readback structure for information from previous tasks*)
	bWriteDataObj : BOOL; (* TRUE=write data object module *)
	bDataObjLenErr : BOOL; (*Error occured in permem: data module size missmatch*)
	bCreateDataObj : BOOL; (* TRUE=create new data object *)
	bWriteOnce : BOOL; (* write permanent memory once *)
	DatObjCreate_01 : DatObjCreate; (* data object create *)
	DatObjInfoBak_02 : DatObjInfo; (* data object info *)
	DatObjDelete_01 : DatObjDelete; (* data object delete *)
	DatObjRead_01 : DatObjRead; (* data object read *)
	DatObjRead_02 : DatObjRead; (* manual initiated data object read *)
	DatObjWrite_01 : DatObjWrite; (* data object write *)
	DatObjDelete_02 : DatObjDelete; (* data object delete *)
	DatObjDelete_11 : DatObjDelete; (*Delete Backup File*)
	DatObjInfo_01 : DatObjInfo; (* data object info *)
	DatObjInfo_02 : DatObjInfo; (* data object info *)
	szModuleName : STRING[35]; (* module name of object *)
	szModuleNameBackup : STRING[35]; (* module name of posiibly created backup object *)
	DatObjCopy_01 : DatObjCopy;
	bCopyDataObj : BOOL;
	TON_WarnDelay : TON;
	TON_WritePMEM : TON; (* delay write permanent memory *)
	ulPMPointer : UDINT; (* adress of actual checksum value *)
	ulChecksum : UDINT; (* parameter checksum value *)
	pm_len : UDINT; (* permanent value lenght *)
	ulChecksumOld : UDINT; (* last vlaue of parameter checksum *)
	ulChkValue : UDINT; (* actual value of parameter pointer *)
	pm_id : UDINT; (* permanent value identifier *)
	pm_p : UDINT; (* permanent value pointer *)
	DatObjInfo_META : DatObjInfo;
	DatObjRead_META : DatObjRead;
	szMetaDataRaw : STRING[2000];
	szMetaData : ARRAY[0..4] OF STRING[35];
	szMetaDataVis : ARRAY[0..3] OF STRING[35];
	ssIndex : INT;
	ssCount : INT;
	ucMetaDataRaw : ARRAY[0..2000] OF USINT;
	ssCount2 : INT;
	szMetaDataFile : STRING[10];
	szText1 : STRING[20];
	pv_adr_IN_XX_tPB2MM : UDINT;
	pv_lng : UDINT;
	pv_lng_IN_XX_tPB2MM : UDINT;
	pv_lng_OUT_XX_tPB2MM : UDINT;
	szText2 : STRING[20];
	pv_adr_OUT_XX_tXX2PB : UDINT;
END_VAR
VAR CONSTANT
	ERR_NOERROR : UINT := 0;
END_VAR
VAR
	usPMWriteCnt : UINT;
	pm_Error : UDINT; (* permanent value error *) (* Deleted: pm : ParaMem_typ; permanent memory tags mathias, 22.8.11*)
	fun_Error : UDINT := 0; (*state > 0 = function error*)
	xLocalParaCheck : ParaCheckFUB; (*local function instance to check parameter values*)
	TON_ParaSetupOk : TON;
	bParaCheckSystemOk : BOOL;
	iDebug_ParaOkChecked : UDINT;
	bRestoreBackupDataObj : BOOL := FALSE;
	bRestoreDataObjContent : BOOL := FALSE;
	pm_id_backup : UDINT;
	pm_p_Backup : UDINT;
	DatObjCopy_02 : DatObjCopy;
	bDeleteBackupDataObj : BOOL := FALSE; (*Command to delete backup data module file on purpose*)
	bDebugPara : ARRAY[0..5] OF BOOL;
	ssIndex2 : INT;
	ssIndex3 : INT;
	ssIndex4 : INT;
	ssIndexVis : INT;
	szText : STRING[40];
	pv_adr_Para : UDINT;
	szParaSnippet : ARRAY[0..5] OF STRING[150];
	szParaIndex : STRING[10];
	slValue : DINT;
	iModuleDLD_ResetCount : INT;
	bDownloadDetected : BOOL;
	bFlagParaStructCopyWorking : BOOL; (*true, if cyclic para copying is active, 1 false cycle at every copy *)
	bStoreInitParaInDataObj : BOOL := FALSE;
	bTestflag : BOOL;
	bReadOutMETA_Once : BOOL;
	tParaCheck_iPvAdress : ARRAY[0..5] OF UDINT;
	tParaCheck_iPvLengt : ARRAY[0..5] OF UDINT;
	tParaCheck_rPvValue : ARRAY[0..5] OF REAL;
	tParaCheck_rRangeMIN : ARRAY[0..5] OF REAL;
	tParaCheck_rRangeMAX : ARRAY[0..5] OF REAL;
	tParaCheck_szPvName : ARRAY[0..5] OF STRING[35];
	ssFormatDetected : INT;
	szMetaDataPart : STRING[150];
	szFullTaskName : STRING[35];
	szFullMetaModuleName : STRING[35];
	debugLen : INT;
	debugSize : INT := 0;
	strcat_adr1 : UDINT;
	strcat_adr2 : UDINT;
	ssIndexTN : INT;
	bAlternate : BOOL;
	n : INT;
	iAlternateChecksum : DINT;
	iAlternateChecksumOld : DINT;
	ulDebugChkValue : ARRAY[0..999] OF UDINT;
	Adr1 : UDINT;
	Adr2 : UDINT;
	usPMWriteCntStepsize : UINT := 1; (*different step sizes to help debug*)
	usPMWriteCntXOR : UINT;
	usPMWriteCntAltSum : UINT;
	ulAdrPM : UDINT;
	usChkValuePM : USINT;
	ulAdrPara : UDINT;
	ulPara_len : UDINT;
	usChkValuePara : USINT;
	iDebugCountPMDifferences : DINT := 0;
	bEngineRunDetected : BOOL; (*detection status bit autocommand 100 /101  for engine run state*)
	ucMetaDataDebugInfoLine : ARRAY[0..24] OF STRING[80];
	ssIndexMand : INT := 0;
	szMetaDataMand : STRING[35];
	iMyErrorInfo_Autoreset : DINT; (*internal autoreset counter*)
	ssIndex_Version : INT; (*internal*)
	ssIndex_BU : INT; (*internal*)
	ssIndex_BU2 : INT; (*internal*)
END_VAR
```

### Package Logical/CBM/PBCMemV2 - Package

### Program Logical/CBM/PBCMemV2/PBC_Control (IEC) - PBC_Control task

#### PBC_Control.st - Cyclic code
```iecst
(*******************************************************************************
AGGR: read and write DIA.NE XT parameter to flash memory	(cyclic)

This code is confidential and proprietary to the INNIO Company.
It may not be used in any form, or reproduced in any manner, without the express
written permission of the INNIO Company.
Copyright, INNIO Company, 2019

Customized modifications: -
------------------------

History:
-------
V3.50		06-06-2014	Caks,		generated
V3.50.1		04-09-2014	Caks,		added: ucPBCBits
V3.50.2		23-10-2014	Caks,		added: auto enable
V3.50.3		05-11-2014	Caks,		added: many new variables
			03-12-2014	Caks,		added: Rod and Main bearing temperature
			05-12-2014	Caks,		added: Time to Structure and File
V3.50.4		12-12-2014	Perktold,   changed activation
V3.50.5		08-01-2015	Perktold,	Änderung Dateinamen
V4.02.0		09-03-2015	Caks,		converted to XT4 CBM module, added some variables
			14-04-2015	Caks,		save Header when triggered
			26-05-2015	Caks,		buffering enabled at 100rpm, write trigger enabled at min 200rpm and added lastcycle bugfix at low rpms
			21-10-2015	Caks,		added SFIKW Event Trigger
V4.02.2		21-08-2017	502423184	Extended version, see spec
V4.06.0		24-04-2018	502423184	new easy way setting up triggers in one line
			30-07-2018	502423184	Bugfix if engine trips in ramp up

Instructions for use:
--------------------

To add ECBMem Triggers --> go to Section 4.3

10ms Task class 1 --> saves every 80ms/120ms the data

Outstandings:
------------
*******************************************************************************)
PROGRAM	_INIT
(** A: ATD Buffer Stopping *)
	TON_MSTOP_10s.PT := T#10s;

END_PROGRAM

PROGRAM _CYCLIC

(** 1: Enable ECBMem on Type 9 Engines or Parameter settings *)
TON_PBCMem_Ena(IN := (NOT(bGnlTrip1 OR bGnlTrip2 OR bGnlTrip3) AND IN_CB.tPB2MM.bParaSetupOk), PT := T#1m);
IF TON_PBCMem_Ena.Q THEN
	bPBC_Mem_Ena	:=	Para.bECBMem_Ena OR xEngType.Type9;
END_IF

(** 2: If enabled do *)
IF bPBC_Mem_Ena THEN

(** 3: ATD Buffer Stopping *)
	TON_MSTOP_10s.IN := xOpMode.Stop;
	TON_MSTOP_10s();
	(*hold the buffer during engine stop to avoid cycle time violation *)
	IF EDGEPOS(bGnlTrip1 OR bGnlTrip2 OR bGnlTrip3) AND NOT bPBC_Write AND NOT xOpMode.Stop THEN
		 bPBC_Write_RStop := TRUE;
	ELSIF TON_MSTOP_10s.Q  THEN
		 bPBC_Write_RStop := FALSE;
	END_IF

(** 4: Triggers *)
(** 4.1: SFIKW & LHE Events *)
	bSFIKW_Event	:=	FALSE;
	FOR i:=1 TO USINT_TO_INT(xEngType.NumberOfCylinder) DO
		bSFIKW_Event	:=	MAX(bSFIKW_Event, IN_CB.bPBCSlowDriftCheck[i]) ;
	END_FOR

(** 4.2: Manual Trigger *)
	IF bPBC_Write OR (VIS2MM.ECB.bTrig AND xOpMode.Stop) OR NOT bPBC_Record THEN						(* disable trigger, if write is performing or in stop mode or not buffering *)
		VIS2MM.ECB.bTrig	:=	FALSE;
	END_IF
	iManCyc	:=	LIMIT(REAL_TO_INT(VIS2MM.ECB.rRemain), -900, 100);

(** 4.3: All Triggers *)
	(* Trigger Name in File 				Remaining cycles after trigger			Trigger bit, on EDGEPOS the trigger is activated, priority from 1 to max *)
	Buffer.TrigMode[1].Name := 'Trip';		Buffer.TrigMode[1].iRemain	:= 0;		Buffer.TrigMode[1].bEvent := Para.bECB_Trig_Alarm AND (bGnlTrip1 OR bGnlTrip2 OR bGnlTrip3);
	Buffer.TrigMode[2].Name := 'LVRT';		Buffer.TrigMode[2].iRemain	:= -300;	Buffer.TrigMode[2].bEvent := Para.bECB_Trig_GC AND IN_CB.bPBC_Event_GC;
	Buffer.TrigMode[3].Name := 'Man';		Buffer.TrigMode[3].iRemain	:= iManCyc;	Buffer.TrigMode[3].bEvent := VIS2MM.ECB.bTrig;
	Buffer.TrigMode[4].Name := 'Misf';		Buffer.TrigMode[4].iRemain	:= 0;		Buffer.TrigMode[4].bEvent := Para.bECB_Trig_Misf AND IN_CB.bPBC_Event_Misf;
	Buffer.TrigMode[5].Name	:= 'SFKW';		Buffer.TrigMode[5].iRemain	:= 0;		Buffer.TrigMode[5].bEvent := Para.bECB_Trig_SFKW AND bSFIKW_Event;
	Buffer.TrigMode[6].Name	:= 'LGM_Ramp';	Buffer.TrigMode[6].iRemain	:= -300;	Buffer.TrigMode[6].bEvent := Para.bECB_Trig_LGM AND bLGM_Event_Ramp;
	Buffer.TrigMode[7].Name	:= 'LGM';		Buffer.TrigMode[7].iRemain	:= -300;	Buffer.TrigMode[7].bEvent := Para.bECB_Trig_LGM AND bLGM_Event;
	Buffer.TrigMode[8].Name := 'IMEP';		Buffer.TrigMode[8].iRemain	:= 0;		Buffer.TrigMode[8].bEvent := FALSE;
	(* Triggers can be here added, don't forget to increase trigger constant --> iECB_MaxTrig *)
	Buffer.TrigMode[9].Name := 'Spare';		Buffer.TrigMode[9].iRemain	:= 0;		Buffer.TrigMode[9].bEvent := FALSE;
	Buffer.TrigMode[10].Name:= 'Spare';		Buffer.TrigMode[10].iRemain	:= 0;		Buffer.TrigMode[10].bEvent:= FALSE;

(** 4.4: Trigger evaluation *)
	bECB_Trigger	:= FALSE;
	FOR i:=1 TO iECB_MaxTrig DO
		IF NOT bECB_Trigger AND Buffer.TrigMode[i].bEvent THEN
			iECB_Trigger	:=	INT_TO_UINT(i);
		END_IF
		bECB_Trigger	:=	bECB_Trigger OR Buffer.TrigMode[i].bEvent;
	END_FOR

(** 5: Action on Trigger Event *)
	IF EDGEPOS(bECB_Trigger) AND NOT bPBC_Write AND NOT xOpMode.Stop AND bPBC_Record THEN
(** 5.1: start last cycles to record *)
		bLast_Cycles	:=	TRUE;
		bPBC_Write		:=	TRUE;
		iPBC_Trigger	:=	iECB_Trigger;
		iLast_Cycles	:=	Buffer.TrigMode[iECB_Trigger].iRemain;

(** 5.2: get Alarms and Warnings *)
		szPBC_Trip_IDs 	:= 	'';
		iCnt_Trip		:=	0;
		szPBC_Warn_IDs 	:= 	'';
		iCnt_Warn		:=	0;
		FOR i:=1001 TO 3999 BY 1 DO												(* go through all relevant error *)
			IF IN_CB.iMsg[i] > 0 AND IN_CB.iMsg[i] < 4 THEN							(* find the active trips *)
				iCnt_Trip	:=	iCnt_Trip + 1;											(* count trips *)
				IF iCnt_Trip < 7 THEN														(* save only 6 nummers = 29 chars *)
					IF iCnt_Trip > 1 THEN 	strcat(ADR(szPBC_Trip_IDs), ADR(';')); END_IF;	(* put between the numbers a ';' *)
	  				itoa(i,ADR(szTemp));	strcat(ADR(szPBC_Trip_IDs), ADR(szTemp));		(* the alarm id's will be saved *)
				END_IF
			END_IF
			IF IN_CB.iMsg[i] = 4 THEN												(* find the active warnings *)
				iCnt_Warn	:=	iCnt_Warn + 1;											(* count warnings *)
				IF iCnt_Warn < 7 THEN														(* save only 6 nummers = 29 chars *)
					IF iCnt_Warn > 1 THEN 	strcat(ADR(szPBC_Warn_IDs), ADR(';')); 	END_IF;	(* put between the numbers a ';' *)
	  				itoa(i,ADR(szTemp));	strcat(ADR(szPBC_Warn_IDs), ADR(szTemp));		(* the warning id's will be saved *)
				END_IF
			END_IF
		END_FOR

(** 5.3: collect header information *)
		iCnt_Header :=	0;
		Buffer.HeaderS[iCnt_Header].Name	:=	'Trigger Delay';
		itoa(100 - iLast_Cycles,ADR(Buffer.HeaderS[iCnt_Header].Value));

		iCnt_Header 						:=	MIN(iCnt_Header + 1, iHS_Max);
		Buffer.HeaderS[iCnt_Header].Name	:=	'Warnings';
		Buffer.HeaderS[iCnt_Header].Value	:=	'';
		Buffer.HeaderS[iCnt_Header].Value	:=	szPBC_Warn_IDs;

		IF bGnlTrip1 OR bGnlTrip2 OR bGnlTrip3  THEN
			iCnt_Header 						:=	MIN(iCnt_Header + 1, iHS_Max);
			Buffer.HeaderS[iCnt_Header].Name	:=	'Trips';
			Buffer.HeaderS[iCnt_Header].Value	:=	'';
			Buffer.HeaderS[iCnt_Header].Value	:=	szPBC_Trip_IDs;
		END_IF

		iCnt_Header 						:=	MIN(iCnt_Header + 1, iHS_Max);
		Buffer.HeaderS[iCnt_Header].Name	:=	'Operation Mode';
		IF xOpMode_old.Idle THEN 			Buffer.HeaderS[iCnt_Header].Value	:=	'Idle';
		ELSIF xOpMode_old.NetP THEN 		Buffer.HeaderS[iCnt_Header].Value	:=	'NetP';
		ELSIF xOpMode_old.Island THEN 		Buffer.HeaderS[iCnt_Header].Value	:=	'Island';
		END_IF

		Buffer.iCnt_HS						:=	iCnt_Header;	//return used size

		//Header 12 Array
		IF Para.bSA_Ign_Active THEN

			iCnt_Header :=	0;
			Buffer.Header12[iCnt_Header].Name	:=	'T_SAFI';
			Buffer.Header12[iCnt_Header].Unit	:=	'degC';
			Buffer.Header12[iCnt_Header].Value	:=	IN_CB.rT_SA_ElecTemp;
			Buffer.Header12[iCnt_Header].Co		:=	1;

			iCnt_Header 						:=	MIN(iCnt_Header + 1, iH12_Max);
			Buffer.Header12[iCnt_Header].Name	:=	'SA_SW_Vers';
			Buffer.Header12[iCnt_Header].Unit	:=	'';
			Buffer.Header12[iCnt_Header].Value	:=	IN_CB.rSA_SW_Vers;
			Buffer.Header12[iCnt_Header].Co		:=	2;

			iCnt_Header 						:=	MIN(iCnt_Header + 1, iH12_Max);
			Buffer.Header12[iCnt_Header].Name	:=	'SA_FiltVers';
			Buffer.Header12[iCnt_Header].Unit	:=	'';
			Buffer.Header12[iCnt_Header].Value	:=	IN_CB.rSA_FiltVers;
			Buffer.Header12[iCnt_Header].Co		:=	2;

			IF Para.bSA_PBC_Active THEN
				iCnt_Header 						:=	MIN(iCnt_Header + 1, iH12_Max);
				Buffer.Header12[iCnt_Header].Name	:=	'Sensor_Sensitivity';
				Buffer.Header12[iCnt_Header].Unit	:=	'mV/bar';
				Buffer.Header12[iCnt_Header].Value	:=	IN_CB.rSA_PBC_Sens;
				Buffer.Header12[iCnt_Header].Co		:=	0;
			END_IF
			Buffer.iCnt_H12						:=	iCnt_Header;	//return used size
		ELSE
			iCnt_Header :=	0;
			Buffer.Header12[iCnt_Header].Name	:=	'no SAFI';
			Buffer.Header12[iCnt_Header].Unit	:=	'';
			Buffer.Header12[iCnt_Header].Value;
			Buffer.Header12[iCnt_Header].Co		:=	1;
			Buffer.iCnt_H12						:=	0;	//return used size
		END_IF

		//Header
		iCnt_Header :=	0;
		Buffer.Header[iCnt_Header].Name		:=	'T_Eng_Oil';
		Buffer.Header[iCnt_Header].Unit		:=	'degC';
		Buffer.Header[iCnt_Header].Value	:=	IN_CB.tT_EO.Unfilt;
		Buffer.Header[iCnt_Header].Co		:=	1;

		iCnt_Header 						:=	MIN(iCnt_Header + 1, iH_Max);
		Buffer.Header[iCnt_Header].Name		:=	'T_Eng_Water';
		Buffer.Header[iCnt_Header].Unit		:=	'degC';
		Buffer.Header[iCnt_Header].Value	:=	IN_CB.tT_ECW.Unfilt;
		Buffer.Header[iCnt_Header].Co		:=	1;

		iCnt_Header 						:=	MIN(iCnt_Header + 1, iH_Max);
		Buffer.Header[iCnt_Header].Name		:=	'T_Amb';
		Buffer.Header[iCnt_Header].Unit		:=	'degC';
		Buffer.Header[iCnt_Header].Value	:=	IN_CB.rT_Ch_T1LP_Avg;
		Buffer.Header[iCnt_Header].Co		:=	1;

		IF IN_CB.tT_GR.Exist THEN
			iCnt_Header 						:=	MIN(iCnt_Header + 1, iH_Max);
			Buffer.Header[iCnt_Header].Name		:=	'T_Gas';
			Buffer.Header[iCnt_Header].Unit		:=	'degC';
			Buffer.Header[iCnt_Header].Value	:=	IN_CB.tT_GR.Unfilt;
			Buffer.Header[iCnt_Header].Co		:=	1;
		END_IF

		iCnt_Header 						:=	MIN(iCnt_Header + 1, iH_Max);
		Buffer.Header[iCnt_Header].Name		:=	'Operating Time';
		Buffer.Header[iCnt_Header].Unit		:=	'h';
		Buffer.Header[iCnt_Header].Value	:=	DINT_TO_REAL(IN_CB.iCnt_OpHours);
		Buffer.Header[iCnt_Header].Co		:=	1;

		iCnt_Header 						:=	MIN(iCnt_Header + 1, iH_Max);
		Buffer.Header[iCnt_Header].Name		:=	'Engine Starts';
		Buffer.Header[iCnt_Header].Unit		:=	'';
		Buffer.Header[iCnt_Header].Value	:=	DINT_TO_REAL(IN_CB.iCnt_Starts);
		Buffer.Header[iCnt_Header].Co		:=	0;

		iCnt_Header 						:=	MIN(iCnt_Header + 1, iH_Max);
		Buffer.Header[iCnt_Header].Name		:=	'P_Nom';
		Buffer.Header[iCnt_Header].Unit		:=	'kW';
		Buffer.Header[iCnt_Header].Value	:=	IN_CB.rP_Nom;
		Buffer.Header[iCnt_Header].Co		:=	0;

		iCnt_Header 						:=	MIN(iCnt_Header + 1, iH_Max);
		Buffer.Header[iCnt_Header].Name		:=	'N_Nom';
		Buffer.Header[iCnt_Header].Unit		:=	'rpm';
		Buffer.Header[iCnt_Header].Value	:=	Para.rN_EngNom;;
		Buffer.Header[iCnt_Header].Co		:=	0;

		IF IN_CB.tPr_Baro.Exist THEN
			iCnt_Header 						:=	MIN(iCnt_Header + 1, iH_Max);
			Buffer.Header[iCnt_Header].Name		:=	'Pr_Baro';
			Buffer.Header[iCnt_Header].Unit		:=	'bar';
			Buffer.Header[iCnt_Header].Value	:=	IN_CB.tPr_Baro.Unfilt;
			Buffer.Header[iCnt_Header].Co		:=	3;
		END_IF

		IF IN_CB.tHumidity_AirIn.Exist THEN
			iCnt_Header 						:=	MIN(iCnt_Header + 1, iH_Max);
			Buffer.Header[iCnt_Header].Name		:=	'Humidity';
			Buffer.Header[iCnt_Header].Unit		:=	'';
			Buffer.Header[iCnt_Header].Value	:=	IN_CB.tHumidity_AirIn.Unfilt;
			Buffer.Header[iCnt_Header].Co		:=	3;
		END_IF

		IF xEngType.Type9 THEN
			iCnt_Header 						:=	MIN(iCnt_Header + 1, iH_Max);
			Buffer.Header[iCnt_Header].Name		:=	'Bal_Coef_a';
			Buffer.Header[iCnt_Header].Unit		:=	'';
			Buffer.Header[iCnt_Header].Value	:=	IN_CB.rPmax_Offset_Coef_a;
			Buffer.Header[iCnt_Header].Co		:=	1;

			iCnt_Header 						:=	MIN(iCnt_Header + 1, iH_Max);
			Buffer.Header[iCnt_Header].Name		:=	'Bal_Coef_b';
			Buffer.Header[iCnt_Header].Unit		:=	'';
			Buffer.Header[iCnt_Header].Value	:=	IN_CB.rPmax_Offset_Coef_b;
			Buffer.Header[iCnt_Header].Co		:=	1;
		END_IF

		iCnt_Header 						:=	MIN(iCnt_Header + 1, iH_Max);
		Buffer.Header[iCnt_Header].Name		:=	'F_Nom';
		Buffer.Header[iCnt_Header].Unit		:=	'Hz';
		Buffer.Header[iCnt_Header].Value	:=	Para.rF_Nom[1];
		Buffer.Header[iCnt_Header].Co		:=	1;

		iCnt_Header 						:=	MIN(iCnt_Header + 1, iH_Max);
		Buffer.Header[iCnt_Header].Name		:=	'I_Nom';
		Buffer.Header[iCnt_Header].Unit		:=	'A';
		Buffer.Header[iCnt_Header].Value	:=	Para.rI_GenNom[1];
		Buffer.Header[iCnt_Header].Co		:=	0;

		iCnt_Header 						:=	MIN(iCnt_Header + 1, iH_Max);
		Buffer.Header[iCnt_Header].Name		:=	'U_Nom';
		Buffer.Header[iCnt_Header].Unit		:=	'V';
		Buffer.Header[iCnt_Header].Value	:=	Para.rU_Gen_Nom[1];
		Buffer.Header[iCnt_Header].Co		:=	0;

		IF xEngType.Type9 THEN
			iCnt_Header 						:=	MIN(iCnt_Header + 1, iH_Max);
			Buffer.Header[iCnt_Header].Name		:=	'Eta_Gen';
			Buffer.Header[iCnt_Header].Unit		:=	'%';
			Buffer.Header[iCnt_Header].Value	:=	IN_CB.rEta_Gen * 100;
			Buffer.Header[iCnt_Header].Co		:=	2;

			iCnt_Header 						:=	MIN(iCnt_Header + 1, iH_Max);
			Buffer.Header[iCnt_Header].Name		:=	'Eta_Mot';
			Buffer.Header[iCnt_Header].Unit		:=	'%';
			Buffer.Header[iCnt_Header].Value	:=	IN_CB.rEta_Eng * 100;
			Buffer.Header[iCnt_Header].Co		:=	2;

			iCnt_Header 						:=	MIN(iCnt_Header + 1, iH_Max);
			Buffer.Header[iCnt_Header].Name		:=	'Eta_Vol';
			Buffer.Header[iCnt_Header].Unit		:=	'%';
			Buffer.Header[iCnt_Header].Value	:=	IN_CB.rVE_Eng * 100;
			Buffer.Header[iCnt_Header].Co		:=	2;
		END_IF

		Buffer.iCnt_H						:=	iCnt_Header;	//return used size

	END_IF

(** 6: Record state machine *)
	IF NOT bPBC_Write AND NOT bPBC_Write_RStop THEN		//start and stop recording when engine turns and during no write event
		bPBC_Record		:=	NOT xOpMode.Stop;
	END_IF
	IF bPBC_Record THEN									//if recorder is activated
		IF bPBC_NewData AND bLast_Cycles THEN				// increase counter if new data is available
			iLast_Cycles := iLast_Cycles + 1;
		END_IF
		IF bLast_Cycles AND (iLast_Cycles >= 100 OR rN_Eng < 1) THEN		// count to 100 and then stop with recording
			bPBC_Record		:=	FALSE;
			bLast_Cycles	:=	FALSE;
			iLast_Cycles	:=	0;
		END_IF
	ELSE
		bLast_Cycles	:=	FALSE;
		iLast_Cycles	:=	0;
	END_IF

(** 7: Clear data from ECBMem buffer in Stop mode *)
	IF EDGEPOS(xOpMode.Stop) THEN
		bClear_Wait		:=	TRUE;
		iSlowDown		:=	0;
	END_IF

	xTON_Clear(IN:= bClear_Wait, PT:=T#40s);	//wait for ATD

	IF xTON_Clear.Q AND NOT bPBC_Record AND NOT bPBC_Write THEN
		(* Reset actual dataset position *)
		iCnt_Cycle		:=	0;
		IF iSlowDown >= 0 AND iSlowDown <= iBufferSize THEN
			iLines := LIMIT(0, iSlowDown, iBufferSize);
			(* Clear Timestamps *)
			Buffer.timer[iLines]							:=	0;
			(* Clear Bits *)
			FOR iData := 0 TO iBits_Max DO
				Buffer.Bits[iData].ucData[iLines]			:=	0;
			END_FOR
			(* Clear Bit Patterns *)
			FOR iData := 0 TO iPC_Max DO
				Buffer.pattern[iData].BitPattern[iLines]	:=	0;
			END_FOR
			(* Clear Engine Cycle Data *)
			FOR iData := 0 TO iEC_Max DO
				Buffer.ui16[iData].Data[iLines]				:=	0;
			END_FOR
			(* Clear Task Cycle Data *)
			FOR iData := 0 TO iTC_Max DO
				Buffer.ui16_H[iData].Hi[iLines]				:=	0;
				Buffer.ui16_H[iData].Lo[iLines]				:=	0;
			END_FOR
		ELSIF iSlowDown > iBufferSize AND iSlowDown <= iBufferSize + iBufferSize10 +1  THEN
			iLines := LIMIT(0, iSlowDown - iBufferSize- 1, iBufferSize10);
			(* Clear Slow Cycle Data *)
			FOR iData := 0 TO iSC_Max DO
				Buffer.ui16_low[iData].Data[iLines] 		:=	0;
			END_FOR
		ELSE
			(* Fertig *)
			bClear_Wait		:=	FALSE;
		END_IF

		(* increase line counter *)
		iSlowDown		:=	iSlowDown + 1;
	END_IF

END_IF

xOpMode_old	:=	xOpMode;

END_PROGRAM
```

#### PBC_Control.var - Local variables
```iecst
(********************************************************************
 * COPYRIGHT -- INNIO Company
 ********************************************************************
 * Program: perm_map
 * File: perm_map.var
 * Author: WaldharM
 * Created: April 05, 2011
 ********************************************************************
 * Local variables of program perm_map
 ********************************************************************)
VAR
	iLast_Cycles : INT;
	bLast_Cycles : BOOL;
	TON_PBCMem_Ena : TON;
	i : INT;
	szTemp : STRING[7];
	iCnt_Warn : INT;
	iCnt_Trip : INT;
	szPBC_Warn_IDs : STRING[31];
	szPBC_Trip_IDs : STRING[31];
	iCnt_Header : INT;
	xOpMode_old : OpMode;
	bSFIKW_Event : BOOL;
	TON_MSTOP_10s : TON := (0);
	bClear_Wait : BOOL := 0;
	iLines : INT;
	iData : INT;
	iSlowDown : INT;
	xTON_Clear : TON := (0);
	iManCyc : INT;
	bECB_Trigger : BOOL := 0;
	iECB_Trigger : UINT;
END_VAR
```

### Program Logical/CBM/PBCMemV2/PBC_Buffer (IEC) - + collectes data every 10ms

- PBC_Buffer.st (not readable text: treated as protected, skipped)

#### PBC_Buffer.var - Local variables
```iecst
(********************************************************************
 * COPYRIGHT -- INNIO Company
 ********************************************************************
 * Program: PBC_Input
 * File: PBC_Input.var
 * Author: 502293141
 * Created: March 11, 2015
 ********************************************************************
 * Local variables of program PBC_Input
 ********************************************************************)
VAR
	GetTC : ARRAY[0..iTC_Max] OF PBC_Lim; (*Task Cycle Class BlackBox*)
	GetEC : ARRAY[0..iEC_Max] OF PBC_In; (*Engine Cycle Class BlackBox*)
	GetSC : ARRAY[0..iSC_Max] OF PBC_In; (*Slow Cycle Class BlackBox*)
	tSkipFire : UDINT;
	szTemp : STRING[5] := '';
	i : INT;
	iCnt : INT;
	iCnt_GetTC : INT;
	iCnt_GetEC : INT;
	iCnt_GetSC : INT;
	ucData : USINT;
	tLimpHome : UDINT;
	tLimpHomeRKS : UDINT;
	tCompLine : UDINT;
	tNegVolt : UDINT;
	tNegPres : UDINT;
	tPresSlope : UDINT;
	tSlowDrift : UDINT;
	tMemBurst : UDINT;
	tSensErr : UDINT;
	tGlowIgn : UDINT;
	tMisf_I : UDINT;
	tMisf_II : UDINT;
	ucData1 : USINT;
	rPr_CPP_Filt_Max : ARRAY[0..24] OF REAL;
	bNOxS_CatOut_Exist : BOOL := 0;
	bNOxS_EngOut_Exist : BOOL := 0;
	bNOxS_EngOut_A_Exist : BOOL := 0;
	bNOxS_EngOut_B_Exist : BOOL := 0;
	tCPSSat : UDINT;
END_VAR
```

#### PBC_Lib.fun
```iecst
(********************************************************************
 * COPYRIGHT -- INNIO Company
 ********************************************************************
 * Program: PBC_MFile
 * File: PBC_MFile.fun
 * Author: 502293141
 * Created: October 27, 2014
 ********************************************************************
 * Functions and function blocks of program PBC_MFile
 ********************************************************************)

FUNCTION_BLOCK PBC_Lim
	VAR_INPUT
		reset : BOOL;
		In : REAL; (*Input*)
		Name : STRING[NameSize]; (*Name max 21 Characters*)
		Store : USINT; (*Determines storage*)
		Unit : STRING[UnitSize]; (*Unit max 5 Characters*)
		Co : REAL; (*Conversion factor 1 = no conversion*)
	END_VAR
	VAR_OUTPUT
		Hi : REAL; (*High*)
		Lo : REAL; (*Low*)
	END_VAR
	VAR
		LCRMinMax_Intern : LCRMinMax;
	END_VAR
END_FUNCTION_BLOCK

FUNCTION_BLOCK PBC_In
	VAR_INPUT
		In : REAL; (*Input*)
		Name : STRING[NameSize]; (*Name max 21 Characters*)
		Store : USINT; (*Determines storage*)
		Unit : STRING[UnitSize]; (*Unit max 5 Characters*)
		Co : REAL; (*Conversion factor 1 = no conversion*)
	END_VAR
	VAR_OUTPUT
		Out : REAL; (*Out*)
	END_VAR
END_FUNCTION_BLOCK
```

### Program Logical/CBM/PBCMemV2/ECB_Test (IEC) - Test Routine for ECB Memory
